// PU2150-03 PUSH DIVERT Extended
PX_4291_Extended(
	In:= In_PX_4291_Extended,
	CFG_OKState:= 0,
	CFG_OnDlyTime:= DebounceOnTime,
	CFG_OnDlyTime:= DebounceOffTime,
	In_Sim:= 
	);

// PU2150-03 PUSH DIVERT Retracted
PX_4311_Retracted(
	In:= In_PX_4311_Retracted,
	CFG_OKState:= 0,
	CFG_OnDlyTime:= DebounceOnTime,
	CFG_OnDlyTime:= DebounceOffTime,
	In_Sim:= 
	);

// PL2140 PLOW DIVERT PISTON PROX Extended
PX_10181_Extended(
	In:= In_PX_10181_Extended,
	CFG_OKState:= 0,
	CFG_OnDlyTime:= DebounceOnTime,
	CFG_OnDlyTime:= DebounceOffTime,
	In_Sim:= 
	);

// PL2140 PLOW DIVERT Extended
PX_10211_Extended(
	In:= In_PX_10211_Extended,
	CFG_OKState:= 0,
	CFG_OnDlyTime:= DebounceOnTime,
	CFG_OnDlyTime:= DebounceOffTime,
	In_Sim:= 
	);

// PL2140 PLOW DIVERT Retracted
PX_10231_Retracted(
	In:= In_PX_10231_Retracted,
	CFG_OKState:= 0,
	CFG_OnDlyTime:= DebounceOnTime,
	CFG_OnDlyTime:= DebounceOffTime,
	In_Sim:= 
	);

// PI2140 PIN STOP Extended
PX_11181_Extended(
	In:= In_PX_11181_Extended,
	CFG_OKState:= 0,
	CFG_OnDlyTime:= DebounceOnTime,
	CFG_OnDlyTime:= DebounceOffTime,
	In_Sim:= 
	);

// PI2140 PIN STOP Retracted
PX_11201_Retracted(
	In:= In_PX_11201_Retracted,
	CFG_OKState:= 0,
	CFG_OnDlyTime:= DebounceOnTime,
	CFG_OnDlyTime:= DebounceOffTime,
	In_Sim:= 
	);

// GR2140-02 "D" GRIPPER Extended
PX_11291_Extended(
	In:= In_PX_11291_Extended,
	CFG_OKState:= 0,
	CFG_OnDlyTime:= DebounceOnTime,
	CFG_OnDlyTime:= DebounceOffTime,
	In_Sim:= 
	);

// GR2140-02 "D" GRIPPER Retracted
PX_11321_Retracted(
	In:= In_PX_11321_Retracted,
	CFG_OKState:= 0,
	CFG_OnDlyTime:= DebounceOnTime,
	CFG_OnDlyTime:= DebounceOffTime,
	In_Sim:= 
	);

// GR2140-01 "D" GRIPPER Extended
PX_11141_Extended(
	In:= In_PX_11141_Extended,
	CFG_OKState:= 0,
	CFG_OnDlyTime:= DebounceOnTime,
	CFG_OnDlyTime:= DebounceOffTime,
	In_Sim:= 
	);

// GR2140-01 "D" GRIPPER Retracted
PX_11161_Retracted(
	In:= In_PX_11161_Retracted,
	CFG_OKState:= 0,
	CFG_OnDlyTime:= DebounceOnTime,
	CFG_OnDlyTime:= DebounceOffTime,
	In_Sim:= 
	);

// P2130 PROX BREAK AWAY Extended
PX_12151_Extended(
	In:= In_PX_12151_Extended,
	CFG_OKState:= 0,
	CFG_OnDlyTime:= DebounceOnTime,
	CFG_OnDlyTime:= DebounceOffTime,
	In_Sim:= 
	);
	
// P3095 PROX BREAK AWAY Extended
PX_12251_Extended(
	In:= In_PX_12251_Extended,
	CFG_OKState:= 0,
	CFG_OnDlyTime:= DebounceOnTime,
	CFG_OnDlyTime:= DebounceOffTime,
	In_Sim:= 
	);

END_PROGRAM

// ---- POUs/Solenoids.TcPOU
PROGRAM Solenoids
VAR
nEquipIndex:	DINT := 0;	// Dummy Equipment Index for Non reporting equipment
//----------------------------------------2140--------------------------------------------------------------
//----------------------------------------GR2140_01--------------------------------------------------------------
   cfgGR2140_01Label:	STRING(20) :=  'GR2140_01';
   cfgGR2140_01ExtendTODetectTime:	TIME := T#5S;
   cfgGR2140_01RetractTODetectTime:	TIME := T#5S;
   GR2140_01			: FB_Solenoid_SA;
   GR2140_01_StatePB	: ST_StateCntrlPB;
	{attribute 'OPC.UA.DA' := '0'}
   GR2140_01_Status	: ST_EquipmentStatus;		// Gripper State 
//----------------------------------------GR2140_02--------------------------------------------------------------
   cfgGR2140_02Label:	STRING(20) :=  'GR2140_02';
   cfgGR2140_02ExtendTODetectTime:	TIME := T#5S;
   cfgGR2140_02RetractTODetectTime:	TIME := T#5S;
   GR2140_02			: FB_Solenoid_SA;
   GR2140_02_StatePB	: ST_StateCntrlPB;
	{attribute 'OPC.UA.DA' := '0'}
   GR2140_02_Status	: ST_EquipmentStatus;		// Gripper State 

//----------------------------------------PI2140_01--------------------------------------------------------------
   cfgPI2140_01Label:	STRING(20) :=  'PI2140_01';
   cfgPI2140_01ExtendTODetectTime:	TIME := T#5S;
   cfgPI2140_01RetractTODetectTime:	TIME := T#5S;
   PI2140_01			: FB_Solenoid_DA;
   PI2140_01_StatePB	: ST_StateCntrlPB;
	{attribute 'OPC.UA.DA' := '0'}
   PI2140_01_Status	: ST_EquipmentStatus;		// Gripper State 

//----------------------------------------PL2140_01--------------------------------------------------------------
   cfgPL2140_01Label:	STRING(20) :=  'PL2140_01';
   cfgPL2140_01ExtendTODetectTime:	TIME := T#5S;
   cfgPL2140_01RetractTODetectTime:	TIME := T#5S;
   PL2140_01			: FB_Solenoid_SA;
   PL2140_01_StatePB	: ST_StateCntrlPB;
	{attribute 'OPC.UA.DA' := '0'}
   PL2140_01_Status	: ST_EquipmentStatus;		// Gripper State 

   
//----------------------------------------2150--------------------------------------------------------------   
//----------------------------------------GR2150_01--------------------------------------------------------------
   cfgGR2150_01Label:	STRING(20) :=  'GR2150_01';
   cfgGR2150_01ExtendTODetectTime:	TIME := T#5S;
   cfgGR2150_01RetractTODetectTime:	TIME := T#5S;
   GR2150_01			: FB_Solenoid_SA;
   GR2150_01_StatePB	: ST_StateCntrlPB;
	{attribute 'OPC.UA.DA' := '0'}
   GR2150_01_Status	: ST_EquipmentStatus;		// Gripper State 

//----------------------------------------PI2150_01--------------------------------------------------------------
   cfgPI2150_01Label:	STRING(20) :=  'PI2150_01';
   cfgPI2150_01ExtendTODetectTime:	TIME := T#5S;
   cfgPI2150_01RetractTODetectTime:	TIME := T#5S;
   PI2150_01			: FB_Solenoid_SA;
   PI2150_01_StatePB	: ST_StateCntrlPB;
	{attribute 'OPC.UA.DA' := '0'}
   PI2150_01_Status	: ST_EquipmentStatus;		// Gripper State 

//----------------------------------------PU2150_01--------------------------------------------------------------
   cfgPU2150_01Label:	STRING(20) :=  'PU2150_01';
   cfgPU2150_01ExtendTODetectTime:	TIME := T#5S;
   cfgPU2150_01RetractTODetectTime:	TIME := T#5S;
   PU2150_01			: FB_Solenoid_SA;
   PU2150_01_StatePB	: ST_StateCntrlPB;
	{attribute 'OPC.UA.DA' := '0'}
   PU2150_01_Status	: ST_EquipmentStatus;		// Gripper State 

//----------------------------------------PU2150_02--------------------------------------------------------------
   cfgPU2150_02Label:	STRING(20) :=  'PU2150_02';
   cfgPU2150_02ExtendTODetectTime:	TIME := T#5S;
   cfgPU2150_02RetractTODetectTime:	TIME := T#5S;
   PU2150_02			: FB_Solenoid_SA;
   PU2150_02_StatePB	: ST_StateCntrlPB;
	{attribute 'OPC.UA.DA' := '0'}
   PU2150_02_Status	: ST_EquipmentStatus;		// Gripper State 

//----------------------------------------PU2150_03--------------------------------------------------------------
   cfgPU2150_03Label:	STRING(20) :=  'PU2150_03';
   cfgPU2150_03ExtendTODetectTime:	TIME := T#5S;
   cfgPU2150_03RetractTODetectTime:	TIME := T#5S;
   PU2150_03			: FB_Solenoid_SA;
   PU2150_03_StatePB	: ST_StateCntrlPB;
	{attribute 'OPC.UA.DA' := '0'}
   PU2150_03_Status	: ST_EquipmentStatus;		// Gripper State 

//----------------------------------------PU2150_04--------------------------------------------------------------
   cfgPU2150_04Label:	STRING(20) :=  'PU2150_04';
   cfgPU2150_04ExtendTODetectTime:	TIME := T#5S;
   cfgPU2150_04RetractTODetectTime:	TIME := T#5S;
   PU2150_04			: FB_Solenoid_SA;
   PU2150_04_StatePB	: ST_StateCntrlPB;
	{attribute 'OPC.UA.DA' := '0'}
   PU2150_04_Status	: ST_EquipmentStatus;		// Gripper State 
END_VAR

VAR PERSISTENT
//----------------------------------------GR2140_01--------------------------------------------------------------
cfgGR2140_01IntlksArry: ARRAY [0..15] OF ST_CfgEvents := [
   (Description := 'Low Air' , DeviceLabel := 'P2140' , OKState := TRUE, StopCode := E_StopCodes.LowAir),
   (Description := 'System Interlocks OK' , DeviceLabel := 'SYSTEM', OKState := TRUE, StopCode := E_StopCodes.SystemStop),
   14(())];
cfgGR2140_01EvntsArry: ARRAY [0..15] OF ST_CfgEvents := [
   (Description := 'Extend To', DeviceLabel := 'GR2140_01', LatchRequired := TRUE, OKState := FALSE, FaultWarn:= TRUE, StopCode := E_StopCodes.ActuatorTO),
   (Description := 'Retract TO', DeviceLabel := 'GR2140_01', LatchRequired := TRUE, FaultWarn:= TRUE, OKState := FALSE, StopCode := E_StopCodes.ActuatorTO),
   (Description := 'System Fault', DeviceLabel := '', OKState := TRUE, FaultWarn:= TRUE, StopCode := E_StopCodes.SystemStop),
   (Description := 'Low Air', DeviceLabel := 'P2140', OKState := TRUE, FaultWarn:= TRUE, StopCode := E_StopCodes.LowAir, EventDelay := T#100MS),
   (Description := 'System Estop', DeviceLabel := 'System', OKState := TRUE, FaultWarn:= TRUE, StopCode := E_StopCodes.SystemStop),
   (Description := 'RIO11171 Comm Fault', DeviceLabel := 'RIO11171', OKState := TRUE, FaultWarn:= TRUE, StopCode := E_StopCodes.FieldIOFLT),
   10(())];
//----------------------------------------GR2140_02--------------------------------------------------------------
cfgGR2140_02IntlksArry: ARRAY [0..15] OF ST_CfgEvents := [
   (Description := 'Low Air' , DeviceLabel := 'P2140' , OKState := TRUE, StopCode := E_StopCodes.LowAir),
   (Description := 'System Interlocks OK' , DeviceLabel := 'SYSTEM', OKState := TRUE, StopCode := E_StopCodes.SystemStop),
   14(())];
cfgGR2140_02EvntsArry: ARRAY [0..15] OF ST_CfgEvents := [
   (Description := 'Extend To', DeviceLabel := 'GR2140_02', LatchRequired := TRUE, OKState := FALSE, FaultWarn:= TRUE, StopCode := E_StopCodes.ActuatorTO),
   (Description := 'Retract TO', DeviceLabel := 'GR2140_02', LatchRequired := TRUE, FaultWarn:= TRUE, OKState := FALSE, StopCode := E_StopCodes.ActuatorTO),
   (Description := 'System Fault', DeviceLabel := '', OKState := TRUE, FaultWarn:= TRUE, StopCode := E_StopCodes.SystemStop),
   (Description := 'Low Air', DeviceLabel := 'P2140', OKState := TRUE, FaultWarn:= TRUE, StopCode := E_StopCodes.LowAir, EventDelay := T#100MS),
   (Description := 'System Estop', DeviceLabel := 'System', OKState := TRUE, FaultWarn:= TRUE, StopCode := E_StopCodes.SystemStop),
   (Description := 'RIO3171 Comm Fault', DeviceLabel := 'RIO3171', OKState := TRUE, FaultWarn:= TRUE, StopCode := E_StopCodes.FieldIOFLT),
   9(())];
//----------------------------------------PI2140_01--------------------------------------------------------------
cfgPI2140_01IntlksArry: ARRAY [0..15] OF ST_CfgEvents := [
   (Description := 'Low Air' , DeviceLabel := 'P2140' , OKState := TRUE, StopCode := E_StopCodes.LowAir),
   (Description := 'System Interlocks OK' , DeviceLabel := 'SYSTEM', OKState := TRUE, StopCode := E_StopCodes.SystemStop),
   14(())];
cfgPI2140_01EvntsArry: ARRAY [0..15] OF ST_CfgEvents := [
   (Description := 'Extend To', DeviceLabel := 'PI2140_01', LatchRequired := TRUE, OKState := FALSE, FaultWarn:= TRUE, StopCode := E_StopCodes.ActuatorTO),
   (Description := 'Retract TO', DeviceLabel := 'PI2140_01', LatchRequired := TRUE, FaultWarn:= TRUE, OKState := FALSE, StopCode := E_StopCodes.ActuatorTO),
   (Description := 'System Fault', DeviceLabel := '', OKState := TRUE, FaultWarn:= TRUE, StopCode := E_StopCodes.SystemStop),
   (Description := 'Low Air', DeviceLabel := 'P2140', OKState := TRUE, FaultWarn:= TRUE, StopCode := E_StopCodes.LowAir, EventDelay := T#100MS),
   10(())];

//----------------------------------------PL2140_01--------------------------------------------------------------
cfgPL2140_01IntlksArry: ARRAY [0..15] OF ST_CfgEvents := [
   (Description := 'Low Air' , DeviceLabel := 'P2140' , OKState := TRUE, StopCode := E_StopCodes.LowAir),
   (Description := 'System Interlocks OK' , DeviceLabel := 'SYSTEM', OKState := TRUE, StopCode := E_StopCodes.SystemStop),
   14(())];
cfgPL2140_01EvntsArry: ARRAY [0..15] OF ST_CfgEvents := [
   (Description := 'Extend To', DeviceLabel := 'PL2140_01', LatchRequired := TRUE, OKState := FALSE, FaultWarn:= TRUE, StopCode := E_StopCodes.ActuatorTO),
   (Description := 'Retract TO', DeviceLabel := 'PL2140_01', LatchRequired := TRUE, FaultWarn:= TRUE, OKState := FALSE, StopCode := E_StopCodes.ActuatorTO),
   (Description := 'System Fault', DeviceLabel := '', OKState := TRUE, FaultWarn:= TRUE, StopCode := E_StopCodes.SystemStop),
   (Description := 'Low Air', DeviceLabel := 'P2140', OKState := TRUE, FaultWarn:= TRUE, StopCode := E_StopCodes.LowAir, EventDelay := T#100MS),
   (Description := 'RIO11171 Comm Fault', DeviceLabel := 'RIO11171', OKState := TRUE, FaultWarn:= TRUE, StopCode := E_StopCodes.FieldIOFLT),
   11(())];
//----------------------------------------GR2150_01--------------------------------------------------------------
cfgGR2150_01IntlksArry: ARRAY [0..15] OF ST_CfgEvents := [
   (Description := 'Low Air' , DeviceLabel := 'P2150' , OKState := TRUE, StopCode := E_StopCodes.LowAir),
   (Description := 'System Interlocks OK' , DeviceLabel := 'SYSTEM', OKState := TRUE, StopCode := E_StopCodes.SystemStop),
   14(())];
cfgGR2150_01EvntsArry: ARRAY [0..15] OF ST_CfgEvents := [
   (Description := 'Extend To', DeviceLabel := '2150_01', LatchRequired := TRUE, OKState := FALSE, FaultWarn:= TRUE, StopCode := E_StopCodes.ActuatorTO),
   (Description := 'Retract TO', DeviceLabel := 'GR2150_01', LatchRequired := TRUE, FaultWarn:= TRUE, OKState := FALSE, StopCode := E_StopCodes.ActuatorTO),
   (Description := 'System Fault', DeviceLabel := '', OKState := TRUE, FaultWarn:= TRUE, StopCode := E_StopCodes.SystemStop),
   (Description := 'Low Air', DeviceLabel := 'P2150', OKState := TRUE, FaultWarn:= TRUE, StopCode := E_StopCodes.LowAir, EventDelay := T#100MS),
   11(())];
//----------------------------------------PI2150_01--------------------------------------------------------------
cfgPI2150_01IntlksArry: ARRAY [0..15] OF ST_CfgEvents := [
   (Description := 'Low Air' , DeviceLabel := 'P2150' , OKState := TRUE, StopCode := E_StopCodes.LowAir),
   (Description := 'System Interlocks OK' , DeviceLabel := 'SYSTEM', OKState := TRUE, StopCode := E_StopCodes.SystemStop),
   14(())];
cfgPI2150_01EvntsArry: ARRAY [0..15] OF ST_CfgEvents := [
   (Description := 'Extend To', DeviceLabel := 'PI2150_01', LatchRequired := TRUE, OKState := FALSE, FaultWarn:= TRUE, StopCode := E_StopCodes.ActuatorTO),
   (Description := 'Retract TO', DeviceLabel := 'PI2150_01', LatchRequired := TRUE, FaultWarn:= TRUE, OKState := FALSE, StopCode := E_StopCodes.ActuatorTO),
   (Description := 'System Fault', DeviceLabel := '', OKState := TRUE, FaultWarn:= TRUE, StopCode := E_StopCodes.SystemStop),
   (Description := 'Low Air', DeviceLabel := 'P2150', OKState := TRUE, FaultWarn:= TRUE, StopCode := E_StopCodes.LowAir, EventDelay := T#100MS),
   11(())];
//----------------------------------------PU2150_01--------------------------------------------------------------
cfgPU2150_01IntlksArry: ARRAY [0..15] OF ST_CfgEvents := [
   (Description := 'Low Air' , DeviceLabel := 'P2150' , OKState := TRUE, StopCode := E_StopCodes.LowAir),
   (Description := 'System Interlocks OK' , DeviceLabel := 'SYSTEM', OKState := TRUE, StopCode := E_StopCodes.SystemStop),
   14(())];
cfgPU2150_01EvntsArry: ARRAY [0..15] OF ST_CfgEvents := [
   (Description := 'Extend To', DeviceLabel := 'PU2150_01', LatchRequired := TRUE, OKState := FALSE, FaultWarn:= TRUE, StopCode := E_StopCodes.ActuatorTO),
   (Description := 'Retract TO', DeviceLabel := 'PU2150_01', LatchRequired := TRUE, FaultWarn:= TRUE, OKState := FALSE, StopCode := E_StopCodes.ActuatorTO),
   (Description := 'System Fault', DeviceLabel := '', OKState := TRUE, FaultWarn:= TRUE, StopCode := E_StopCodes.SystemStop),
   (Description := 'Low Air', DeviceLabel := 'P2150', OKState := TRUE, FaultWarn:= TRUE, StopCode := E_StopCodes.LowAir, EventDelay := T#100MS),
   (Description := 'RIO3171 Comm Fault', DeviceLabel := 'RIO3171', OKState := TRUE, FaultWarn:= TRUE, StopCode := E_StopCodes.FieldIOFLT),
   10(())];
//----------------------------------------PU2150_02--------------------------------------------------------------
cfgPU2150_02IntlksArry: ARRAY [0..15] OF ST_CfgEvents := [
   (Description := 'Low Air' , DeviceLabel := 'P2150' , OKState := TRUE, StopCode := E_StopCodes.LowAir),
   (Description := 'System Interlocks OK' , DeviceLabel := 'SYSTEM', OKState := TRUE, StopCode := E_StopCodes.SystemStop),
   14(())];
cfgPU2150_02EvntsArry: ARRAY [0..15] OF ST_CfgEvents := [
   (Description := 'Extend To', DeviceLabel := 'PU2150_02', LatchRequired := TRUE, OKState := FALSE, FaultWarn:= TRUE, StopCode := E_StopCodes.ActuatorTO),
   (Description := 'Retract TO', DeviceLabel := 'PU2150_02', LatchRequired := TRUE, FaultWarn:= TRUE, OKState := FALSE, StopCode := E_StopCodes.ActuatorTO),
   (Description := 'System Fault', DeviceLabel := '', OKState := TRUE, FaultWarn:= TRUE, StopCode := E_StopCodes.SystemStop),
   (Description := 'Low Air', DeviceLabel := 'P2150', OKState := TRUE, FaultWarn:= TRUE, StopCode := E_StopCodes.LowAir, EventDelay := T#100MS),
   (Description := 'RIO3171 Comm Fault', DeviceLabel := 'RIO3171', OKState := TRUE, FaultWarn:= TRUE, StopCode := E_StopCodes.FieldIOFLT),
   10(())];
//----------------------------------------PU2150_03--------------------------------------------------------------
cfgPU2150_03IntlksArry: ARRAY [0..15] OF ST_CfgEvents := [
   (Description := 'Low Air' , DeviceLabel := 'P2150' , OKState := TRUE, StopCode := E_StopCodes.LowAir),
   (Description := 'System Interlocks OK' , DeviceLabel := 'SYSTEM', OKState := TRUE, StopCode := E_StopCodes.SystemStop),
   14(())];
cfgPU2150_03EvntsArry: ARRAY [0..15] OF ST_CfgEvents := [
   (Description := 'Extend To', DeviceLabel := 'PU2150_03', LatchRequired := TRUE, OKState := FALSE, FaultWarn:= TRUE, StopCode := E_StopCodes.ActuatorTO),
   (Description := 'Retract TO', DeviceLabel := 'PU2150_03', LatchRequired := TRUE, FaultWarn:= TRUE, OKState := FALSE, StopCode := E_StopCodes.ActuatorTO),
   (Description := 'System Fault', DeviceLabel := '', OKState := TRUE, FaultWarn:= TRUE, StopCode := E_StopCodes.SystemStop),
   (Description := 'Low Air', DeviceLabel := 'P2150', OKState := TRUE, FaultWarn:= TRUE, StopCode := E_StopCodes.LowAir, EventDelay := T#100MS),
   (Description := 'RIO4141 Comm Fault', DeviceLabel := 'RIO4141', OKState := TRUE, FaultWarn:= TRUE, StopCode := E_StopCodes.FieldIOFLT),
   10(())];
//----------------------------------------PU2150_04--------------------------------------------------------------
cfgPU2150_04IntlksArry: ARRAY [0..15] OF ST_CfgEvents := [
   (Description := 'Low Air' , DeviceLabel := 'P2150' , OKState := TRUE, StopCode := E_StopCodes.LowAir),
   (Description := 'System Interlocks OK' , DeviceLabel := 'SYSTEM', OKState := TRUE, StopCode := E_StopCodes.SystemStop),
   14(())];
cfgPU2150_04EvntsArry: ARRAY [0..15] OF ST_CfgEvents := [
   (Description := 'Extend To', DeviceLabel := 'PU2150_04', LatchRequired := TRUE, OKState := FALSE, FaultWarn:= TRUE, StopCode := E_StopCodes.ActuatorTO),
   (Description := 'Retract TO', DeviceLabel := 'PU2150_04', LatchRequired := TRUE, FaultWarn:= TRUE, OKState := FALSE, StopCode := E_StopCodes.ActuatorTO),
   (Description := 'System Fault', DeviceLabel := '', OKState := TRUE, FaultWarn:= TRUE, StopCode := E_StopCodes.SystemStop),
   (Description := 'Low Air', DeviceLabel := 'P2150', OKState := TRUE, FaultWarn:= TRUE, StopCode := E_StopCodes.LowAir, EventDelay := T#100MS),
   (Description := 'RIO4141 Comm Fault', DeviceLabel := 'RIO4141', OKState := TRUE, FaultWarn:= TRUE, StopCode := E_StopCodes.FieldIOFLT),
   10(())];	
END_VAR

// REMOVE THIS!!!!!!
GVL_IO.SystemAirPressure := TRUE;
//----------------------------------------2140--------------------------------------------------------------
//----------------------------------------GR2140_01--------------------------------------------------------------
GR2140_01_StatePB.AutoPB := System.Cnvyr_Auto;
GR2140_01_StatePB.ManPB := System.Cnvyr_Manual;
GR2140_01_StatePB.ResetPB := System.Cnvyr_Reset;
GR2140_01_StatePB.OfflinePB := System.Cnvyr_Offline;
GR2140_01_StatePB.StopPB := System.Cnvyr_Manual;

// Initialize the Equipment Type
GR2140_01_Status.Sts_EquipmentState.EquipType := E_EquipType.Gripper_SA;

// Interlocks
GR2140_01.In_EquipIntlks.0:= GVL_IO.SystemAirPressure;
//Events
GR2140_01.In_EquipEvents.2:= SystemSafety.Safety_SystemEstopsOK;
GR2140_01.In_EquipEvents.3:= GVL_IO.SystemAirPressure;
GR2140_01.In_EquipEvents.4:= SystemSafety.Safety_SystemEstopsOK;
GR2140_01.In_EquipEvents.5:= NOT CommStatus.RIO11171_CommFault.Out;

// Function Call
GR2140_01(
   In_p_EquipStatePB:= GR2140_01_StatePB,
   In_SimActive:= System.Sys_SimActive,
   In_EquipInit:= GVL_IO.INIT,
   Cfg_UseExtedFdbc:=FALSE,
   In_P_SVReqExtend:= Singulation_Control.SortSingulation_P2140.Out_Grabber_1_Ext,
   In_EquipRtrcdFdbck := ProxSensors.PX_11161_Retracted.Out,
   In_EquipExtdFdbck := ProxSensors.PX_11141_Extended.Out,
   Cfg_EquipIndex := nEquipIndex,
   Cfg_EquipLabel := cfgGR2140_01Label,
   Cfg_EquipDefState:= System.ConvDefaultState,
   Cfg_EquipIntlksArry:= cfgGR2140_01IntlksArry,
   Cfg_EquipEvntsArry:= cfgGR2140_01EvntsArry,
   Cfg_ExtendDetectTime:= cfgGR2140_01ExtendTODetectTime,
   Cfg_RetractDetectTime:= cfgGR2140_01RetractTODetectTime,
   Sts_EquipState := GR2140_01_Status,
   Out_ExtendCrntSV => GVL_IO.GR2140_01_Extend);
//----------------------------------------GR2140_02--------------------------------------------------------------
GR2140_02_StatePB.AutoPB := System.Cnvyr_Auto;
GR2140_02_StatePB.ManPB := System.Cnvyr_Manual;
GR2140_02_StatePB.ResetPB := System.Cnvyr_Reset;
GR2140_02_StatePB.OfflinePB := System.Cnvyr_Offline;
GR2140_02_StatePB.StopPB := System.Cnvyr_Manual;

// Initialize the Equipment Type
GR2140_02_Status.Sts_EquipmentState.EquipType := E_EquipType.Gripper_SA;

// Interlocks
GR2140_02.In_EquipIntlks.0:= GVL_IO.SystemAirPressure;
//Events
GR2140_02.In_EquipEvents.2:= SystemSafety.Safety_SystemEstopsOK;
GR2140_02.In_EquipEvents.3:= GVL_IO.SystemAirPressure;
GR2140_02.In_EquipEvents.4:= SystemSafety.Safety_SystemEstopsOK;
GR2140_02.In_EquipEvents.5:= NOT CommStatus.RIO11171_CommFault.Out;

// Function Call
GR2140_02(
   In_p_EquipStatePB:= GR2140_02_StatePB,
   In_SimActive:= System.Sys_SimActive,
   In_EquipInit:= GVL_IO.INIT,
   Cfg_UseExtedFdbc:=FALSE,
   In_P_SVReqExtend:= Singulation_Control.SortSingulation_P2140.Out_Grabber_2_Ext,
   In_EquipRtrcdFdbck := ProxSensors.PX_11321_Retracted.Out,
   In_EquipExtdFdbck := ProxSensors.PX_11291_Extended.Out,
   Cfg_EquipIndex := nEquipIndex,
   Cfg_EquipLabel := cfgGR2140_02Label,
   Cfg_EquipDefState:= System.ConvDefaultState,
   Cfg_EquipIntlksArry:= cfgGR2140_02IntlksArry,
   Cfg_EquipEvntsArry:= cfgGR2140_02EvntsArry,
   Cfg_ExtendDetectTime:= cfgGR2140_02ExtendTODetectTime,
   Cfg_RetractDetectTime:= cfgGR2140_02RetractTODetectTime,
   Sts_EquipState := GR2140_02_Status,
   Out_ExtendCrntSV => GVL_IO.GR2140_02_Extend); 
//----------------------------------------PI2140_01--------------------------------------------------------------
PI2140_01_StatePB.AutoPB := System.Cnvyr_Auto;
PI2140_01_StatePB.ManPB := System.Cnvyr_Manual;
PI2140_01_StatePB.ResetPB := System.Cnvyr_Reset;
PI2140_01_StatePB.OfflinePB := System.Cnvyr_Offline;
PI2140_01_StatePB.StopPB := System.Cnvyr_Manual;

// Initialize the Equipment Type
PI2140_01_Status.Sts_EquipmentState.EquipType := E_EquipType.Gripper_DA;

// Interlocks
//PI2140_01.In_EquipIntlks.0:= GVL_IO.SystemAirPressure;
// Interlocks for downstream full when the pin stop is extended
PI2140_01.In_EquipIntlks.2:= Photoeyes.PE_8141.Out_OnOffFltrd AND ProxSensors.PX_11181_Extended.Out;
PI2140_01.In_EquipIntlks.3:= Photoeyes.PE_4161.Out_OnOffFltrd AND ProxSensors.PX_11181_Extended.Out;
//Events
PI2140_01.In_EquipEvents.2:= SystemSafety.Safety_SystemEstopsOK;
PI2140_01.In_EquipEvents.3:= GVL_IO.SystemAirPressure;
PI2140_01.In_EquipEvents.4:= SystemSafety.Safety_SystemEstopsOK;
PI2140_01.In_EquipEvents.5:= NOT CommStatus.RIO11171_CommFault.Out;

// Function Call
PI2140_01(
   In_p_EquipStatePB:= PI2140_01_StatePB,
   In_SimActive:= System.Sys_SimActive,
   In_EquipInit:= GVL_IO.INIT,
   In_P_SVReqExtend:= Singulation_Control.SortSingulation_P2140.Out_PinStop_Ext,
   In_P_SVReqRetract:= Singulation_Control.SortSingulation_P2140.Out_PinStop_Ret,
   In_EquipRtrcdFdbck := ProxSensors.PX_11201_Retracted.Out,
   In_EquipExtdFdbck := ProxSensors.PX_11181_Extended.Out,
   Cfg_EquipIndex := nEquipIndex,
   Cfg_EquipLabel := cfgPI2140_01Label,
   Cfg_EquipDefState:= System.ConvDefaultState,   Cfg_EquipIntlksArry:= cfgPI2140_01IntlksArry,
   Cfg_EquipEvntsArry:= cfgPI2140_01EvntsArry,
   Cfg_ExtendDetectTime:= cfgPI2140_01ExtendTODetectTime,
   Cfg_RetractDetectTime:= cfgPI2140_01RetractTODetectTime,
   Sts_EquipState := PI2140_01_Status,
   Out_ExtendCrntSV => GVL_IO.PI2140_01_Extend,  
   Out_RetractCrntSV => GVL_IO.PI2140_01_Retract); 
 
//----------------------------------------PL2140_01--------------------------------------------------------------
PL2140_01_StatePB.AutoPB := System.Cnvyr_Auto;
PL2140_01_StatePB.ManPB := System.Cnvyr_Manual;
PL2140_01_StatePB.ResetPB := System.Cnvyr_Reset;
PL2140_01_StatePB.OfflinePB := System.Cnvyr_Offline;
PL2140_01_StatePB.StopPB := System.Cnvyr_Manual;

// Initialize the Equipment Type
PL2140_01_Status.Sts_EquipmentState.EquipType := E_EquipType.Gripper_SA;

// Interlocks
//PL2140_01.In_EquipIntlks.0:= GVL_IO.SystemAirPressure;
PL2140_01.In_EquipIntlks.2:= Photoeyes.PE_8141.Out_OnOffFltrd;
PL2140_01.In_EquipIntlks.3:= Photoeyes.PE_4161.Out_OnOffFltrd;
//Events
PL2140_01.In_EquipEvents.2:= SystemSafety.Safety_SystemEstopsOK;
PL2140_01.In_EquipEvents.3:= GVL_IO.SystemAirPressure;
PL2140_01.In_EquipEvents.4:= SystemSafety.Safety_SystemEstopsOK;
PL2140_01.In_EquipEvents.5:= NOT CommStatus.RIO10161_CommFault.Out;
PL2140_01.In_EquipIntlks.6:= Photoeyes.PE_10151.JamDetected;

// Function Call
PL2140_01(
   In_p_EquipStatePB:= PL2140_01_StatePB,
   In_SimActive:= System.Sys_SimActive,
   In_EquipInit:= GVL_IO.INIT,
   In_P_SVReqExtend:= Sorter.aSorterDiverts_P2140[1].Output1,
   In_EquipRtrcdFdbck := ProxSensors.PX_10231_Retracted.Out,
   In_EquipExtdFdbck := ProxSensors.PX_10211_Extended.Out,
   Cfg_EquipIndex := nEquipIndex,
   Cfg_EquipLabel := cfgPL2140_01Label,
   Cfg_EquipDefState:= System.ConvDefaultState,
   Cfg_EquipIntlksArry:= cfgPL2140_01IntlksArry,
   Cfg_EquipEvntsArry:= cfgPL2140_01EvntsArry,
   Cfg_ExtendDetectTime:= cfgPL2140_01ExtendTODetectTime,
   Cfg_RetractDetectTime:= cfgPL2140_01RetractTODetectTime,
   Sts_EquipState := PL2140_01_Status,
   Out_ExtendCrntSV => GVL_IO.PL2140_01_Extend); 
//----------------------------------------GR2150_01--------------------------------------------------------------
GR2150_01_StatePB.AutoPB := System.Cnvyr_Auto;
GR2150_01_StatePB.ManPB := System.Cnvyr_Manual;
GR2150_01_StatePB.ResetPB := System.Cnvyr_Reset;
GR2150_01_StatePB.OfflinePB := System.Cnvyr_Offline;
GR2150_01_StatePB.StopPB := System.Cnvyr_Manual;

// Initialize the Equipment Type
GR2150_01_Status.Sts_EquipmentState.EquipType := E_EquipType.Gripper_SA;

// Interlocks
GR2150_01.In_EquipIntlks.0:= GVL_IO.SystemAirPressure;
//Events
GR2150_01.In_EquipEvents.2:= SystemSafety.Safety_SystemEstopsOK;
GR2150_01.In_EquipEvents.3:= GVL_IO.SystemAirPressure;
GR2150_01.In_EquipEvents.4:= SystemSafety.Safety_SystemEstopsOK;
PI2150_01.In_EquipEvents.5:= NOT CommStatus.RIO3171_CommFault.Out;

// Function Call
GR2150_01(
   In_p_EquipStatePB:= GR2150_01_StatePB,
   In_SimActive:= System.Sys_SimActive,
   In_EquipInit:= GVL_IO.INIT,
   Cfg_UseExtedFdbc:=FALSE,
   In_P_SVReqExtend:= Singulation_Control.SortSingulation_P2150.Out_Grabber_1_Ext,
   In_EquipRtrcdFdbck := ProxSensors.PX_2201_Retracted.Out,
   In_EquipExtdFdbck := ProxSensors.PX_2181_Extended.Out,
   Cfg_EquipIndex := nEquipIndex,
   Cfg_EquipLabel := cfgGR2150_01Label,
   Cfg_EquipDefState:= System.ConvDefaultState,
   Cfg_EquipIntlksArry:= cfgGR2150_01IntlksArry,
   Cfg_EquipEvntsArry:= cfgGR2150_01EvntsArry,
   Cfg_ExtendDetectTime:= cfgGR2150_01ExtendTODetectTime,
   Cfg_RetractDetectTime:= cfgGR2150_01RetractTODetectTime,
   Sts_EquipState := GR2150_01_Status,
   Out_ExtendCrntSV => GVL_IO.GR2150_01_Extend); 
//----------------------------------------PI2150_01--------------------------------------------------------------
PI2150_01_StatePB.AutoPB := System.Cnvyr_Auto;
PI2150_01_StatePB.ManPB := System.Cnvyr_Manual;
PI2150_01_StatePB.ResetPB := System.Cnvyr_Reset;
PI2150_01_StatePB.OfflinePB := System.Cnvyr_Offline;
PI2150_01_StatePB.StopPB := System.Cnvyr_Manual;

// Initialize the Equipment Type
PI2150_01_Status.Sts_EquipmentState.EquipType := E_EquipType.Gripper_SA;

// Interlocks
PI2150_01.In_EquipIntlks.0:= GVL_IO.SystemAirPressure;
//Events
PI2150_01.In_EquipEvents.2:= SystemSafety.Safety_SystemEstopsOK;
PI2150_01.In_EquipEvents.3:= GVL_IO.SystemAirPressure;
PI2150_01.In_EquipEvents.4:= SystemSafety.Safety_SystemEstopsOK;
PI2150_01.In_EquipEvents.5:= NOT CommStatus.RIO3171_CommFault.Out;

// Function Call
PI2150_01(
   In_p_EquipStatePB:= PI2150_01_StatePB,
   In_SimActive:= System.Sys_SimActive,
   In_EquipInit:= GVL_IO.INIT,
   In_P_SVReqExtend:= Singulation_Control.SortSingulation_P2150.Out_PinStop_Ext,
   In_EquipRtrcdFdbck := ProxSensors.PX_2151_Retracted.Out,
   In_EquipExtdFdbck := ProxSensors.PX_2131_Extended.Out,
   Cfg_EquipIndex := nEquipIndex,
   Cfg_EquipLabel := cfgPI2150_01Label,
   Cfg_EquipDefState:= System.ConvDefaultState,
   Cfg_EquipIntlksArry:= cfgPI2150_01IntlksArry,
   Cfg_EquipEvntsArry:= cfgPI2150_01EvntsArry,
   Cfg_ExtendDetectTime:= cfgPI2150_01ExtendTODetectTime,
   Cfg_RetractDetectTime:= cfgPI2150_01RetractTODetectTime,
   Sts_EquipState := PI2150_01_Status,
   Out_ExtendCrntSV => GVL_IO.PI2150_01_Extend); 
//----------------------------------------PU2150_01--------------------------------------------------------------
PU2150_01_StatePB.AutoPB := System.Cnvyr_Auto;
PU2150_01_StatePB.ManPB := System.Cnvyr_Manual;
PU2150_01_StatePB.ResetPB := System.Cnvyr_Reset;
PU2150_01_StatePB.OfflinePB := System.Cnvyr_Offline;
PU2150_01_StatePB.StopPB := System.Cnvyr_Manual;

// Initialize the Equipment Type
PU2150_01_Status.Sts_EquipmentState.EquipType := E_EquipType.Gripper_SA;

// Interlocks
PU2150_01.In_EquipIntlks.0:= GVL_IO.SystemAirPressure;
//Events
PU2150_01.In_EquipEvents.2:= SystemSafety.Safety_SystemEstopsOK;
PU2150_01.In_EquipEvents.3:= GVL_IO.SystemAirPressure;
PU2150_01.In_EquipEvents.4:= SystemSafety.Safety_SystemEstopsOK;
PU2150_01.In_EquipEvents.5:= NOT CommStatus.RIO3171_CommFault.Out;

// Function Call
PU2150_01(
   In_p_EquipStatePB:= PU2150_01_StatePB,
   In_SimActive:= System.Sys_SimActive,
   In_EquipInit:= GVL_IO.INIT,
   In_P_SVReqExtend:= Sorter.aSorterDiverts_P2150[1].Output1,
   In_EquipRtrcdFdbck := ProxSensors.PX_3331_Retracted.Out,
   In_EquipExtdFdbck := ProxSensors.PX_3301_Extended.Out,
   Cfg_EquipIndex := nEquipIndex,
   Cfg_EquipLabel := cfgPU2150_01Label,
   Cfg_EquipDefState:= System.ConvDefaultState,
   Cfg_EquipIntlksArry:= cfgPU2150_01IntlksArry,
   Cfg_EquipEvntsArry:= cfgPU2150_01EvntsArry,
   Cfg_ExtendDetectTime:= cfgPU2150_01ExtendTODetectTime,
   Cfg_RetractDetectTime:= cfgPU2150_01RetractTODetectTime,
   Sts_EquipState := PU2150_01_Status,
   Out_ExtendCrntSV => GVL_IO.PU2150_01_Extend); 
//----------------------------------------PU2150_02--------------------------------------------------------------
PU2150_02_StatePB.AutoPB := System.Cnvyr_Auto;
PU2150_02_StatePB.ManPB := System.Cnvyr_Manual;
PU2150_02_StatePB.ResetPB := System.Cnvyr_Reset;
PU2150_02_StatePB.OfflinePB := System.Cnvyr_Offline;
PU2150_02_StatePB.StopPB := System.Cnvyr_Manual;

// Initialize the Equipment Type
PU2150_02_Status.Sts_EquipmentState.EquipType := E_EquipType.Gripper_SA;

// Interlocks
PU2150_02.In_EquipIntlks.0:= GVL_IO.SystemAirPressure;
//Events
PU2150_02.In_EquipEvents.2:= SystemSafety.Safety_SystemEstopsOK;
PU2150_02.In_EquipEvents.3:= GVL_IO.SystemAirPressure;
PU2150_02.In_EquipEvents.4:= SystemSafety.Safety_SystemEstopsOK;
PU2150_02.In_EquipEvents.5:= NOT CommStatus.RIO3171_CommFault.Out;

// Function Call
PU2150_02(
   In_p_EquipStatePB:= PU2150_02_StatePB,
   In_SimActive:= System.Sys_SimActive,
   In_EquipInit:= GVL_IO.INIT,
   In_P_SVReqExtend:= Sorter.aSorterDiverts_P2150[2].Output1,
   In_EquipRtrcdFdbck := ProxSensors.PX_3191_Retracted.Out,
   In_EquipExtdFdbck := ProxSensors.PX_3171_Extended.Out,
   Cfg_EquipIndex := nEquipIndex,
   Cfg_EquipLabel := cfgPU2150_02Label,
   Cfg_EquipDefState:= System.ConvDefaultState,
   Cfg_EquipIntlksArry:= cfgPU2150_02IntlksArry,
   Cfg_EquipEvntsArry:= cfgPU2150_02EvntsArry,
   Cfg_ExtendDetectTime:= cfgPU2150_02ExtendTODetectTime,
   Cfg_RetractDetectTime:= cfgPU2150_02RetractTODetectTime,
   Sts_EquipState := PU2150_02_Status,
   Out_ExtendCrntSV => GVL_IO.PU2150_02_Extend); 
//----------------------------------------PU2150_03--------------------------------------------------------------
PU2150_03_StatePB.AutoPB := System.Cnvyr_Auto;
PU2150_03_StatePB.ManPB := System.Cnvyr_Manual;
PU2150_03_StatePB.ResetPB := System.Cnvyr_Reset;
PU2150_03_StatePB.OfflinePB := System.Cnvyr_Offline;
PU2150_03_StatePB.StopPB := System.Cnvyr_Manual;

// Initialize the Equipment Type
PU2150_03_Status.Sts_EquipmentState.EquipType := E_EquipType.Gripper_SA;

// Interlocks
PU2150_03.In_EquipIntlks.0:= GVL_IO.SystemAirPressure;
//Events
PU2150_03.In_EquipEvents.2:= SystemSafety.Safety_SystemEstopsOK;
PU2150_03.In_EquipEvents.3:= GVL_IO.SystemAirPressure;
PU2150_03.In_EquipEvents.4:= SystemSafety.Safety_SystemEstopsOK;
PU2150_03.In_EquipEvents.5:= NOT CommStatus.RIO4141_CommFault.Out;

// Function Call
PU2150_03(
   In_p_EquipStatePB:= PU2150_03_StatePB,
   In_SimActive:= System.Sys_SimActive,
   In_EquipInit:= GVL_IO.INIT,
   In_P_SVReqExtend:= Sorter.aSorterDiverts_P2150[3].Output1,
   In_EquipRtrcdFdbck := ProxSensors.PX_4311_Retracted.Out,
   In_EquipExtdFdbck := ProxSensors.PX_4291_Extended.Out,
   Cfg_EquipIndex := nEquipIndex,
   Cfg_EquipLabel := cfgPU2150_03Label,
   Cfg_EquipDefState:= System.ConvDefaultState,
   Cfg_EquipIntlksArry:= cfgPU2150_03IntlksArry,
   Cfg_EquipEvntsArry:= cfgPU2150_03EvntsArry,
   Cfg_ExtendDetectTime:= cfgPU2150_03ExtendTODetectTime,
   Cfg_RetractDetectTime:= cfgPU2150_03RetractTODetectTime,
   Sts_EquipState := PU2150_03_Status,
   Out_ExtendCrntSV => GVL_IO.PU2150_03_Extend);
//----------------------------------------PU2150_04--------------------------------------------------------------
PU2150_04_StatePB.AutoPB := System.Cnvyr_Auto;
PU2150_04_StatePB.ManPB := System.Cnvyr_Manual;
PU2150_04_StatePB.ResetPB := System.Cnvyr_Reset;
PU2150_04_StatePB.OfflinePB := System.Cnvyr_Offline;
PU2150_04_StatePB.StopPB := System.Cnvyr_Manual;

// Initialize the Equipment Type
PU2150_04_Status.Sts_EquipmentState.EquipType := E_EquipType.Gripper_SA;

// Interlocks
PU2150_04.In_EquipIntlks.0:= GVL_IO.SystemAirPressure;
//Events
PU2150_04.In_EquipEvents.2:= SystemSafety.Safety_SystemEstopsOK;
PU2150_04.In_EquipEvents.3:= GVL_IO.SystemAirPressure;
PU2150_04.In_EquipEvents.4:= SystemSafety.Safety_SystemEstopsOK;
PU2150_04.In_EquipEvents.5:= NOT CommStatus.RIO4141_CommFault.Out;

// Function Call
PU2150_04(
   In_p_EquipStatePB:= PU2150_04_StatePB,
   In_SimActive:= System.Sys_SimActive,
   In_EquipInit:= GVL_IO.INIT,
   In_P_SVReqExtend:= Sorter.aSorterDiverts_P2150[4].Output1,
   In_EquipRtrcdFdbck := ProxSensors.PX_4171_Retracted.Out,
   In_EquipExtdFdbck := ProxSensors.PX_4151_Extended.Out,
   Cfg_EquipIndex := nEquipIndex,
   Cfg_EquipLabel := cfgPU2150_04Label,
   Cfg_EquipDefState:= System.ConvDefaultState,
   Cfg_EquipIntlksArry:= cfgPU2150_04IntlksArry,
   Cfg_EquipEvntsArry:= cfgPU2150_04EvntsArry,
   Cfg_ExtendDetectTime:= cfgPU2150_04ExtendTODetectTime,
   Cfg_RetractDetectTime:= cfgPU2150_04RetractTODetectTime,
   Sts_EquipState := PU2150_04_Status,
   Out_ExtendCrntSV => GVL_IO.PU2150_04_Extend);

END_PROGRAM

// ---- FunctionBlocks/Solenoids/Functions/FB_Solenoid_SA.TcPOU
FUNCTION_BLOCK FB_Solenoid_SA

(* Single-Acting solenoid Set up,
	Uses Interlocks. No common interlocks
	Doesn't use Start Conditions or the horn delay  
	Uses Events and has 5 that can be uassigned that are location specific and a common events for the Actuator Extended/Retracted Time-out faults 

	Regardless of the travel of the actuator, the following define the extended and retracted positions
		Extended is the position expected when the solenoid valve is actuated
		Retracted is the position expected when the solenoid valve is resting
*)

VAR_IN_OUT
	CFG_EquipIndex				: DINT;	// Index used for local Equipment status array
	{attribute 'OPC.UA.DA' := '1'}
	Sts_EquipState					: ST_EquipmentStatus;		// State Status
//	In_EquipEvents					: UINT;		// Event that is specific to the instance of the solenoid/actuator
//	In_EquipIntlks					: UINT;		// Interlock that is specific to the instance of the solenoid/actuator
END_VAR
VAR_INPUT
	{attribute 'OPC.UA.DA' := '1'}
	In_o_EquipStatePB				: ST_StateCntrlPB;		// Hmi push buttons to change states
	In_p_EquipStatePB				: ST_StateCntrlPB;		// programming to change states
	In_P_SVReqExtend			: BOOL;		// Input to extend actuator if in auto and conditions are met
	In_SimActive				: BOOL;
	In_EquipInit					: BOOL;		// Initialise;
	{attribute 'OPC.UA.DA' := '1'}
	In_EquipExtdFdbck			: BOOL := FALSE;	// Actuator Extended Feedback (1 = Extended)
	{attribute 'OPC.UA.DA' := '1'}
	In_EquipRtrcdFdbck			: BOOL := FALSE;	// Actuator Retracted Feedback (1 = Retracted)
	Cfg_EquipDefState				: E_StateCntrl;
	{attribute 'OPC.UA.DA' := '1'}
	Cfg_EquipLabel					: STRING(20);		// Label of the Solenoid
	Cfg_UseExtedFdbc			: BOOL := FALSE;	// Use Feedback from actuator for Extended state, otherwise, use output 

	// Events
	In_EquipEvents					: UINT;		// Event that is specific to the instance of the solenoid/actuator
	
	{attribute 'OPC.UA.DA' := '0'}
	Cfg_EquipEvntsArry				: ARRAY [0..15] OF ST_CfgEvents;
	Cfg_ExtendDetectTime		: TIME;
	Cfg_RetractDetectTime		: TIME;
	
	// Interlocks that can be Instance Specific
	In_EquipIntlks					: UINT;		// Interlock that is specific to the instance of the solenoid/actuator
	{attribute 'OPC.UA.DA' := '0'}
	Cfg_EquipIntlksArry			: ARRAY [0..15] OF ST_CfgEvents;		// Descriptions of the Interlock 
	
END_VAR
VAR_OUTPUT
	{attribute 'OPC.UA.DA' := '1'}
	Out_ExtendCrntSV			: BOOL;		// Extend command for the current solenoid/actuator
	{attribute 'OPC.UA.DA' := '1'}
	Sts_ExtendCrntSV			: BOOL;		// Status showing that current solenoid/actuator is extended/extending
	{attribute 'OPC.UA.DA' := '1'}
	Sts_All_Intlks_OK			: BOOL;		// Status bit to show that all interloks are good to Run 
	{attribute 'OPC.UA.DA' := '1'}
	Sts_FaultActive				: BOOL;	// Status Bit Showing that a fault is present (0= No Active Faults, 1= Fault Active)
	{attribute 'OPC.UA.DA' := '1'}
	Sts_WarnActive				: BOOL;	// Status Bit Showing that a warning is present (0= No Active Warnings, 1= Warning Active)
	{attribute 'OPC.UA.DA' := '1'}
	Sts_All_Evnts_OK			: BOOL;		// Status Bit Showing that ALL Events are OK to RUN (0= Event Present, 1= OK to Run)
	{attribute 'OPC.UA.DA' := '1'}
	Sts_IntlksArry				: ARRAY[0..15] OF ST_EventSts;		// Interlock status 0 to 15 Input
	{attribute 'OPC.UA.DA' := '1'}
	Sts_FaultsArry				: ARRAY[0..15] OF ST_EventSts;	// Status of each Fault Event State (0= OFF, 1=ON)
	{attribute 'OPC.UA.DA' := '1'}
	Sts_WarnsArry				: ARRAY[0..15] OF ST_EventSts;		// Status of each Warning Event State (0= OFF, 1=ON)
	{attribute 'OPC.UA.DA' := '0'}
	Sts_EvntsArry				: ARRAY[0..15] OF ST_EventSts; 	// Status of each Event State (0= OFF, 1=ON)
END_VAR
VAR
	{attribute 'OPC.UA.DA' := '0'}
	SV_fbIntrlks				: FB_Intlks_Latch;
	SV_IntlksArry				: ARRAY[0..15] OF BOOL;
	{attribute 'OPC.UA.DA' := '0'}
	SV_fbEquipCntrl				: FB_EquipCntrl;
	{attribute 'OPC.UA.DA' := '0'}
	SV_EventManager				: FB_EventMngr;
	SV_ExtendFault				: FB_JamDetect;			// This FB can also detect when it takes to long to extend an actuator
	SV_RetractFault				: FB_JamDetect;			// This FB can also detect when it takes to long to retract an actuator
	SV_EventArry				: ARRAY[0..15] OF BOOL;
	
	SV_LatchIgnore				: BOOL := FALSE;		// Put as a place holder for ease of future use
	SV_LatchReset				: BOOL := FALSE;		//Put as a place holder for ease of future use
	SV_IntlkBypassed			: ARRAY [0..15] OF BOOL;		//Put as a place holder for ease of future use
	SV_MoveEnabled				: BOOL;					// TRUE = Enable the SV/Actuator to operate
	SV_StartEnabled				: BOOL;					// TRUE = Start Motion for SV/actuator

END_VAR

// Set Up Common Single-Acting solenoid Interlocks and inputs for interlocks that are specific for the configuration instance
SV_IntlksArry[0] := In_EquipIntlks.0;
SV_IntlksArry[1] := System.SysIntlksAllOk; 
SV_IntlksArry[2] := In_EquipIntlks.2;
SV_IntlksArry[3] := In_EquipIntlks.3;
SV_IntlksArry[4] := In_EquipIntlks.4;
SV_IntlksArry[5] := In_EquipIntlks.5;
SV_IntlksArry[6] := In_EquipIntlks.6;
SV_IntlksArry[7] := In_EquipIntlks.7;
SV_IntlksArry[8] := In_EquipIntlks.8;
SV_IntlksArry[9] := In_EquipIntlks.9; 
SV_IntlksArry[10] := In_EquipIntlks.10;
SV_IntlksArry[11] := In_EquipIntlks.11;
SV_IntlksArry[12] := In_EquipIntlks.12;
SV_IntlksArry[13] := In_EquipIntlks.13;
SV_IntlksArry[14] := In_EquipIntlks.14;
SV_IntlksArry[15] := In_EquipIntlks.15;

In_EquipIntlks:=0;
	
// Call Interlock block
SV_fbIntrlks(
	In_Intlks:= SV_IntlksArry,
	CFG_IntlksArry:= Cfg_EquipIntlksArry, 
	HMI_LatchIgnore:= SV_LatchIgnore, 
	HMI_LatchReset:= SV_LatchReset, 
	All_Intlk_OK=> Sts_All_Intlks_OK, 
	STS_Intlks=> Sts_IntlksArry);
	
// Set Up Common Solenoid Events and inputs for events that are specific for the configuration instance
SV_EventArry[0]:= SV_ExtendFault.JamDetected;	// Even though this is a JamDetected output, it is really a Extend time-out fault
SV_EventArry[1]:= SV_RetractFault.JamDetected;	// Even though this is a JamDetected output, it is really a retract time-out fault
SV_EventArry[2]:= In_EquipEvents.2;
SV_EventArry[3]:= In_EquipEvents.3;
SV_EventArry[4]:= In_EquipEvents.4;
SV_EventArry[5]:= In_EquipEvents.5;
SV_EventArry[6]:= In_EquipEvents.6;
SV_EventArry[7]:= In_EquipEvents.7;
SV_EventArry[8]:= In_EquipEvents.8;
SV_EventArry[9]:= In_EquipEvents.9;
SV_EventArry[10]:= In_EquipEvents.10;
SV_EventArry[11]:= In_EquipEvents.11;
SV_EventArry[12]:= In_EquipEvents.12;
SV_EventArry[13]:= In_EquipEvents.13;
SV_EventArry[14]:= In_EquipEvents.14;
SV_EventArry[15]:= In_EquipEvents.15;

//In_EquipEvents:=0;

// Event Manager
SV_EventManager(
	sEquipStateCntrlSts := Sts_EquipState.Sts_EquipmentState,
	In_EventsArry := SV_EventArry ,  
	CFG_EvntsArry:= Cfg_EquipEvntsArry, 
	HMI_LatchReset:= In_o_EquipStatePB.ResetPB OR In_p_EquipStatePB.ResetPB,
	Out_FaultActive=> Sts_FaultActive, 
	Out_WarnActive=> Sts_WarnActive, 
	Sts_All_Evnts_OK=> Sts_All_Evnts_OK, 
	Sts_FaultsArry=> Sts_FaultsArry, 
	Sts_WarnsArry=> Sts_WarnsArry, 
	Sts_EvntsArry=> Sts_EvntsArry);
	
(*
	Set up individual Events that are common for this configuration
 	For the Extend Fault, use one of two conditions
		1 - If the SV is configured to use Extended feedback, check the input
		2 - If the SV is not configured to use Extedned feedback, check that the output is on and the retracted input is not on
*)
SV_ExtendFault.In_PE := ((Cfg_UseExtedFdbc AND NOT In_EquipExtdFdbck)
					OR (NOT Cfg_UseExtedFdbc AND (Out_ExtendCrntSV AND In_EquipRtrcdFdbck)))
					AND NOT Sts_EquipState.Sts_EquipmentState.StsOffline
					AND NOT In_o_EquipStatePB.ResetPB
					AND NOT In_p_EquipStatePB.ResetPB;
SV_ExtendFault(
	In_Status:= Out_ExtendCrntSV,
	CFG_PEOKState:= 0, 
	JamDetTime:= cfg_ExtendDetectTime);
	
(*
 	For the Retract Fault, use the following condition
		Output is off and the actuator is not in the retracted condition
*)
SV_RetractFault.In_PE := NOT Out_ExtendCrntSV
					AND NOT In_EquipRtrcdFdbck
					AND NOT Sts_EquipState.Sts_EquipmentState.StsOffline
					AND NOT In_o_EquipStatePB.ResetPB
					AND NOT In_p_EquipStatePB.ResetPB;
SV_RetractFault(
	In_Status:= NOT Out_ExtendCrntSV,
	CFG_PEOKState:= 0, 
	JamDetTime:= cfg_RetractDetectTime);

//Call Equipment FB to control current SV/Actuator	
SV_fbEquipCntrl(
	CFG_EquipIndex := cfg_EquipIndex,
	CFG_EquipLabel := Cfg_EquipLabel,
	CFG_UseStrtCnd:= FALSE, 
	CFG_UseIntrlks:= TRUE, 
	CFG_UseHrnDly:= FALSE, 
	CFG_EquipDefState:= Cfg_EquipDefState, 
	In_IntlksOK:= Sts_All_Intlks_OK, 
	In_SimActive:= In_SimActive, 
	In_Init:= In_EquipInit, 
	o_EquipStatePB:= In_o_EquipStatePB, 
	p_EquipStatePB:= In_p_EquipStatePB, 
	P_EquipReqRun:= In_P_SVReqExtend, 
	In_EquipFaults:= Sts_FaultActive, 
	Out_EquipRun=> , 
	Out_Horn=> , 
	Sts_EquipState:= Sts_EquipState.Sts_EquipmentState);	

// Process the SV_MoveEnabled signal
SV_MoveEnabled := SV_fbEquipCntrl.Out_EquipRun;

SV_StartEnabled := SV_MoveEnabled;	

// Actuate the SV based on the results of the Equipment Control state
IF Sts_EquipState.Sts_EquipmentState.CrntState = E_StateCntrl.stAuto THEN
	IF (In_P_SVReqExtend )
	   THEN
		Out_ExtendCrntSV := SV_StartEnabled;
		// Set Solenoid Actuation Status
		Sts_ExtendCrntSV := (Out_ExtendCrntSV) OR (In_SimActive AND SV_fbEquipCntrl.RunApproved);
	ELSE
		Out_ExtendCrntSV := FALSE;
		// Set Solenoid Actuation Status
		Sts_ExtendCrntSV := FALSE;
	END_IF
ELSE
	IF (In_o_EquipStatePB.ManExtendPB)
	   THEN
		Out_ExtendCrntSV := SV_StartEnabled;
		// Set Solenoid Actuation Status
		Sts_ExtendCrntSV := (Out_ExtendCrntSV) OR (In_SimActive AND SV_fbEquipCntrl.RunApproved);
	ELSE
		Out_ExtendCrntSV := FALSE;
		// Set Solenoid Actuation Status
		Sts_ExtendCrntSV := FALSE;
	END_IF
END_IF

// Turn OFF Extend and Retract when a stop is issued
IF In_p_EquipStatePB.StopPB OR In_o_EquipStatePB.StopPB OR Sts_FaultActive THEN
	Out_ExtendCrntSV := FALSE;
	Sts_ExtendCrntSV := FALSE;
END_IF

// Capture the Operation state of the Solenoid/actuator
IF Sts_ExtendCrntSV THEN
	// Solenoid Actuating/Entending
	Sts_EquipState.Sts_EquipmentState.CrntOperState := E_OperStateCntrl.extending;
	// Solenoid Extended
	IF (Cfg_UseExtedFdbc AND In_EquipExtdFdbck) OR (NOT Cfg_UseExtedFdbc AND (Out_ExtendCrntSV AND NOT In_EquipRtrcdFdbck)) THEN
		Sts_EquipState.Sts_EquipmentState.CrntOperState := E_OperStateCntrl.extended;
	END_IF
ELSE
	// Solenoid Retracting
	Sts_EquipState.Sts_EquipmentState.CrntOperState := E_OperStateCntrl.retracting;
	// Solenoid Retracted
	IF In_EquipRtrcdFdbck THEN
		Sts_EquipState.Sts_EquipmentState.CrntOperState := E_OperStateCntrl.retracted;
	END_IF
END_IF
IF NOT Sts_ExtendCrntSV
   AND NOT In_EquipRtrcdFdbck
   AND NOT (Cfg_UseExtedFdbc AND In_EquipExtdFdbck) OR (NOT Cfg_UseExtedFdbc AND (Out_ExtendCrntSV AND NOT In_EquipRtrcdFdbck)) 
   THEN
	Sts_EquipState.Sts_EquipmentState.CrntOperState := E_OperStateCntrl.unknown;
END_IF
// Solenoid control and state
CASE Sts_EquipState.Sts_EquipmentState.CrntOperState OF
	E_OperStateCntrl.extended:
			Sts_EquipState.Sts_IsExtended := TRUE;
			Sts_EquipState.Sts_IsExtending := FALSE;
			Sts_EquipState.Sts_IsRetracted := FALSE;
			Sts_EquipState.Sts_IsRetracting := FALSE;
	E_OperStateCntrl.extending:
			Sts_EquipState.Sts_IsExtended := FALSE;
			Sts_EquipState.Sts_IsExtending := TRUE;
			Sts_EquipState.Sts_IsRetracted := FALSE;
			Sts_EquipState.Sts_IsRetracting := FALSE;
	E_OperStateCntrl.retracted:
			Sts_EquipState.Sts_IsExtended := FALSE;
			Sts_EquipState.Sts_IsExtending := FALSE;
			Sts_EquipState.Sts_IsRetracted := TRUE;
			Sts_EquipState.Sts_IsRetracting := FALSE;
	E_OperStateCntrl.retracting:
			Sts_EquipState.Sts_IsExtended := FALSE;
			Sts_EquipState.Sts_IsExtending := FALSE;
			Sts_EquipState.Sts_IsRetracted := FALSE;
			Sts_EquipState.Sts_IsRetracting := TRUE;
END_CASE

// Populate the Sts Output Variables
Sts_EquipState.Sts_All_Intlks_OK  := Sts_All_Intlks_OK;
Sts_EquipState.Sts_All_Evnts_OK  := Sts_All_Evnts_OK;
Sts_EquipState.Sts_FaultActive := Sts_FaultActive;
Sts_EquipState.Sts_WarnActive := Sts_WarnActive;

END_FUNCTION_BLOCK

// ---- FunctionBlocks/Solenoids/Functions/FB_Solenoid_DA.TcPOU
FUNCTION_BLOCK FB_Solenoid_DA

(* Double-Acting solenoid Set up,
	Uses Interlocks. No common interlocks
	Doesn't use Start Conditions or the horn delay  
	Uses Events and has 5 that can be uassigned that are location specific and a common events for the Actuator Extended/Retracted Time-out faults 

	Regardless of the travel of the actuator, the following define the extended and retracted positions
		Extended is the position expected when the solenoid valve is actuated
		Retracted is the position expected when the solenoid valve is resting
*)

VAR_IN_OUT
	CFG_EquipIndex				: DINT;	// Index used for local Equipment status array
	{attribute 'OPC.UA.DA' := '1'}
	Sts_EquipState					: ST_EquipmentStatus;		// State Status
//	In_EquipEvents					: UINT;		// Event that is specific to the instance of the solenoid/actuator
//	In_EquipIntlks					: UINT;		// Interlock that is specific to the instance of the solenoid/actuator
END_VAR
VAR_INPUT
	{attribute 'OPC.UA.DA' := '1'}
	In_o_EquipStatePB				: ST_StateCntrlPB;		// Hmi push buttons to change states
	In_p_EquipStatePB				: ST_StateCntrlPB;		// programming to change states
	In_P_SVReqExtend			: BOOL;		// Input to extend actuator if in auto and conditions are met
	In_P_SVReqRetract			: BOOL;		// Input to retract actuator if in auto and conditions are met
	In_SimActive				: BOOL;
	In_EquipInit					: BOOL;		// Initialise;
	{attribute 'OPC.UA.DA' := '1'}
	In_EquipExtdFdbck			: BOOL := FALSE;	// Actuator Extended Feedback (1 = Extended)
	{attribute 'OPC.UA.DA' := '1'}
	In_EquipRtrcdFdbck			: BOOL := FALSE;	// Actuator Retracted Feedback (1 = Retracted)
	Cfg_EquipDefState				: E_StateCntrl;
	{attribute 'OPC.UA.DA' := '1'}
	Cfg_EquipLabel					: STRING(20);		// Label of the Solenoid
	Cfg_UseExtedFdbc			: BOOL := FALSE;	// Use Feedback from actuator for Extended state, otherwise, use output 

	// Events
	// This is the system interlock, but could be something different
	In_EquipEvents					: UINT;		// Event that is specific to the instance of the solenoid/actuator
	
	{attribute 'OPC.UA.DA' := '0'}
	Cfg_EquipEvntsArry				: ARRAY [0..15] OF ST_CfgEvents;
	Cfg_ExtendDetectTime		: TIME;
	Cfg_RetractDetectTime		: TIME;
	
	// Interlocks that can be Instance Specific
	In_EquipIntlks					: UINT;		// Interlock that is specific to the instance of the solenoid/actuator
	{attribute 'OPC.UA.DA' := '0'}
	Cfg_EquipIntlksArry			: ARRAY [0..15] OF ST_CfgEvents;		// Descriptions of the Interlock 
	
END_VAR
VAR_OUTPUT
	{attribute 'OPC.UA.DA' := '1'}
	Out_ExtendCrntSV			: BOOL;		// Extend command for the current solenoid/actuator
	{attribute 'OPC.UA.DA' := '1'}
	Sts_ExtendCrntSV			: BOOL;		// Status showing that current solenoid/actuator is extended/extending
	{attribute 'OPC.UA.DA' := '1'}
	Out_RetractCrntSV			: BOOL;		// Retract command for the current solenoid/actuator
	{attribute 'OPC.UA.DA' := '1'}
	Sts_RetractCrntSV			: BOOL;		// Status showing that current solenoid/actuator is retracteded/retractinging
	{attribute 'OPC.UA.DA' := '1'}
	Sts_All_Intlks_OK			: BOOL;		// Status bit to show that all interloks are good to Run 
	{attribute 'OPC.UA.DA' := '1'}
	Sts_FaultActive				: BOOL;	// Status Bit Showing that a fault is present (0= No Active Faults, 1= Fault Active)
	{attribute 'OPC.UA.DA' := '1'}
	Sts_WarnActive				: BOOL;	// Status Bit Showing that a warning is present (0= No Active Warnings, 1= Warning Active)
	{attribute 'OPC.UA.DA' := '1'}
	Sts_All_Evnts_OK			: BOOL;		// Status Bit Showing that ALL Events are OK to RUN (0= Event Present, 1= OK to Run)
	{attribute 'OPC.UA.DA' := '1'}
	Sts_IntlksArry				: ARRAY[0..15] OF ST_EventSts;		// Interlock status 0 to 15 Input
	{attribute 'OPC.UA.DA' := '1'}
	Sts_FaultsArry				: ARRAY[0..15] OF ST_EventSts;	// Status of each Fault Event State (0= OFF, 1=ON)
	{attribute 'OPC.UA.DA' := '1'}
	Sts_WarnsArry				: ARRAY[0..15] OF ST_EventSts;		// Status of each Warning Event State (0= OFF, 1=ON)
	{attribute 'OPC.UA.DA' := '0'}
	Sts_EvntsArry				: ARRAY[0..15] OF ST_EventSts; 	// Status of each Event State (0= OFF, 1=ON)
END_VAR
VAR
	{attribute 'OPC.UA.DA' := '0'}
	SV_fbIntrlks				: FB_Intlks_Latch;
	SV_IntlksArry				: ARRAY[0..15] OF BOOL;
	{attribute 'OPC.UA.DA' := '0'}
	SV_fbEquipCntrl				: FB_EquipCntrl;
	{attribute 'OPC.UA.DA' := '0'}
	SV_EventManager				: FB_EventMngr;
	SV_ExtendFault				: FB_JamDetect;			// This FB can also detect when it takes to long to extend an actuator
	SV_RetractFault				: FB_JamDetect;			// This FB can also detect when it takes to long to retract an actuator
	SV_EventArry				: ARRAY[0..15] OF BOOL;
	
	SV_LatchIgnore				: BOOL := FALSE;		// Put as a place holder for ease of future use
	SV_LatchReset				: BOOL := FALSE;		//Put as a place holder for ease of future use
	SV_IntlkBypassed			: ARRAY [0..15] OF BOOL;		//Put as a place holder for ease of future use
	SV_MoveEnabled				: BOOL;					// TRUE = Enable the SV/Actuator to operate
	SV_StartEnabled				: BOOL;					// TRUE = Start Motion for SV/actuator

END_VAR

// Set Up Common Single-Acting solenoid Interlocks and inputs for interlocks that are specific for the configuration instance
SV_IntlksArry[0] := In_EquipIntlks.0;
SV_IntlksArry[1] := System.SysIntlksAllOk; 
SV_IntlksArry[2] := In_EquipIntlks.2;
SV_IntlksArry[3] := In_EquipIntlks.3;
SV_IntlksArry[4] := In_EquipIntlks.4;
SV_IntlksArry[5] := In_EquipIntlks.5;
SV_IntlksArry[6] := In_EquipIntlks.6;
SV_IntlksArry[7] := In_EquipIntlks.7;
SV_IntlksArry[8] := In_EquipIntlks.8;
SV_IntlksArry[9] := In_EquipIntlks.9; 
SV_IntlksArry[10] := In_EquipIntlks.10;
SV_IntlksArry[11] := In_EquipIntlks.11;
SV_IntlksArry[12] := In_EquipIntlks.12;
SV_IntlksArry[13] := In_EquipIntlks.13;
SV_IntlksArry[14] := In_EquipIntlks.14;
SV_IntlksArry[15] := In_EquipIntlks.15;
	
In_EquipIntlks:= 0;

// Call Interlock block
SV_fbIntrlks(
	In_Intlks:= SV_IntlksArry,
	CFG_IntlksArry:= Cfg_EquipIntlksArry, 
	HMI_LatchIgnore:= SV_LatchIgnore, 
	HMI_LatchReset:= SV_LatchReset, 
	All_Intlk_OK=> Sts_All_Intlks_OK, 
	STS_Intlks=> Sts_IntlksArry);
	
// Set Up Common Solenoid Events and inputs for events that are specific for the configuration instance
SV_EventArry[0]:= SV_ExtendFault.JamDetected;	// Even though this is a JamDetected output, it is really a Extend time-out fault
SV_EventArry[1]:= SV_RetractFault.JamDetected;	// Even though this is a JamDetected output, it is really a retract time-out fault
SV_EventArry[2]:= In_EquipEvents.2;
SV_EventArry[3]:= In_EquipEvents.3;
SV_EventArry[4]:= In_EquipEvents.4;
SV_EventArry[5]:= In_EquipEvents.5;
SV_EventArry[6]:= In_EquipEvents.6;
SV_EventArry[7]:= In_EquipEvents.7;
SV_EventArry[8]:= In_EquipEvents.8;
SV_EventArry[9]:= In_EquipEvents.9;
SV_EventArry[10]:= In_EquipEvents.10;
SV_EventArry[11]:= In_EquipEvents.11;
SV_EventArry[12]:= In_EquipEvents.12;
SV_EventArry[13]:= In_EquipEvents.13;
SV_EventArry[14]:= In_EquipEvents.14;
SV_EventArry[15]:= In_EquipEvents.15;

//In_EquipEvents:=0;

// Event Manager
SV_EventManager(
	sEquipStateCntrlSts := Sts_EquipState.Sts_EquipmentState,
	In_EventsArry := SV_EventArry ,  
	CFG_EvntsArry:= Cfg_EquipEvntsArry, 
	HMI_LatchReset:= In_o_EquipStatePB.ResetPB OR In_p_EquipStatePB.ResetPB,
	Out_FaultActive=> Sts_FaultActive, 
	Out_WarnActive=> Sts_WarnActive, 
	Sts_All_Evnts_OK=> Sts_All_Evnts_OK, 
	Sts_FaultsArry=> Sts_FaultsArry, 
	Sts_WarnsArry=> Sts_WarnsArry, 
	Sts_EvntsArry=> Sts_EvntsArry);
	
(*
	Set up individual Events that are common for this configuration
 	For the Extend Fault, use one of two conditions
		1 - If the SV is configured to use Extended feedback, check the input
		2 - If the SV is not configured to use Extedned feedback, check that the output is on and the retracted input is not on
*)
SV_ExtendFault.In_PE := ((Cfg_UseExtedFdbc AND NOT In_EquipExtdFdbck)
					OR (NOT Cfg_UseExtedFdbc AND (Out_ExtendCrntSV AND In_EquipRtrcdFdbck)))
					AND NOT Sts_EquipState.Sts_EquipmentState.StsOffline
					AND NOT In_o_EquipStatePB.ResetPB
					AND NOT In_p_EquipStatePB.ResetPB;
SV_ExtendFault(
	In_Status:= Out_ExtendCrntSV,
	CFG_PEOKState:= 0, 
	JamDetTime:= cfg_ExtendDetectTime);
	
(*
 	For the Retract Fault, use the following condition
		Retracted Output is ON and the actuator is not in the retracted condition
*)
SV_RetractFault.In_PE := Out_RetractCrntSV
				AND NOT In_EquipRtrcdFdbck
				AND NOT Sts_EquipState.Sts_EquipmentState.StsOffline
				AND NOT In_o_EquipStatePB.ResetPB
				AND NOT In_p_EquipStatePB.ResetPB;
SV_RetractFault(
	In_Status:= Out_RetractCrntSV,
	CFG_PEOKState:= 0, 
	JamDetTime:= cfg_RetractDetectTime);

//Call Equipment FB to control current SV/Actuator	
// XOR the Extend and Retract. The interlocks/events must be prefixed with the extend or retract command 
SV_fbEquipCntrl(
	CFG_EquipIndex := cfg_EquipIndex,
	CFG_EquipLabel := Cfg_EquipLabel,
	CFG_UseStrtCnd:= FALSE, 
	CFG_UseIntrlks:= TRUE, 
	CFG_UseHrnDly:= FALSE, 
	CFG_EquipDefState:= Cfg_EquipDefState, 
	In_IntlksOK:= Sts_All_Intlks_OK, 
	In_SimActive:= In_SimActive, 
	In_Init:= In_EquipInit, 
	o_EquipStatePB:= In_o_EquipStatePB, 
	p_EquipStatePB:= In_p_EquipStatePB, 
	P_EquipReqRun:= In_P_SVReqExtend XOR In_P_SVReqRetract, 
	In_EquipFaults:= Sts_FaultActive, 
	Out_EquipRun=> , 
	Out_Horn=> , 
	Sts_EquipState:= Sts_EquipState.Sts_EquipmentState);	

// Process the SV_MoveEnabled signal
SV_MoveEnabled := SV_fbEquipCntrl.Out_EquipRun;

SV_StartEnabled := SV_MoveEnabled;	

// Actuate the SV based on the results of the Equipment Control state
IF Sts_EquipState.Sts_EquipmentState.CrntState = E_StateCntrl.stAuto THEN
	IF (In_P_SVReqExtend AND NOT In_P_SVReqRetract)
	   THEN
		Out_RetractCrntSV := FALSE;
		Out_ExtendCrntSV := SV_StartEnabled;
		// Set Solenoid Actuation Status
		Sts_ExtendCrntSV := (Out_ExtendCrntSV) OR (In_SimActive AND SV_fbEquipCntrl.RunApproved);
		Sts_RetractCrntSV := FALSE;
	END_IF
	IF In_P_SVReqRetract THEN
		Out_RetractCrntSV := SV_StartEnabled;
		Out_ExtendCrntSV := FALSE;
		// Set Solenoid Actuation Status
		Sts_RetractCrntSV := (Out_RetractCrntSV) OR (In_SimActive AND SV_fbEquipCntrl.RunApproved);
		Sts_ExtendCrntSV := FALSE;
	END_IF
ELSE
	IF (In_o_EquipStatePB.ManExtendPB AND NOT In_o_EquipStatePB.ManRetractPB)
	   THEN
		Out_RetractCrntSV := FALSE;
		Out_ExtendCrntSV := SV_StartEnabled;
		// Set Solenoid Actuation Status
		Sts_ExtendCrntSV := (Out_ExtendCrntSV) OR (In_SimActive AND SV_fbEquipCntrl.RunApproved);
		Sts_RetractCrntSV := FALSE;
	END_IF
	IF In_o_EquipStatePB.ManRetractPB THEN
		Out_RetractCrntSV := SV_StartEnabled;
		Out_ExtendCrntSV := FALSE;
		// Set Solenoid Actuation Status
		Sts_RetractCrntSV := (Out_RetractCrntSV) OR (In_SimActive AND SV_fbEquipCntrl.RunApproved);
		Sts_ExtendCrntSV := FALSE;
	END_IF
END_IF

// Turn OFF Extend and Retract when a stop is issued
IF In_p_EquipStatePB.StopPB OR In_o_EquipStatePB.StopPB OR Sts_FaultActive THEN
	Out_ExtendCrntSV := FALSE;
	Out_RetractCrntSV := FALSE;
	Sts_ExtendCrntSV := FALSE;
	Sts_RetractCrntSV := FALSE;
END_IF

// Capture the Operation state of the Solenoid/actuator
IF Sts_ExtendCrntSV THEN
	// Solenoid Actuating/Entending
	Sts_EquipState.Sts_EquipmentState.CrntOperState := E_OperStateCntrl.extending;
	// Solenoid Extended
	IF (Cfg_UseExtedFdbc AND In_EquipExtdFdbck) OR (NOT Cfg_UseExtedFdbc AND (Out_ExtendCrntSV AND NOT In_EquipRtrcdFdbck)) THEN
		Sts_EquipState.Sts_EquipmentState.CrntOperState := E_OperStateCntrl.extended;
	END_IF
END_IF
IF Sts_RetractCrntSV THEN
	// Solenoid Retracting
	Sts_EquipState.Sts_EquipmentState.CrntOperState := E_OperStateCntrl.retracting;
	// Solenoid Retracted
	IF In_EquipRtrcdFdbck THEN
		Sts_EquipState.Sts_EquipmentState.CrntOperState := E_OperStateCntrl.retracted;
	END_IF
END_IF
IF NOT Sts_ExtendCrntSV
   AND NOT Sts_RetractCrntSV 
   AND NOT In_EquipRtrcdFdbck
   AND NOT (Cfg_UseExtedFdbc AND In_EquipExtdFdbck) OR (NOT Cfg_UseExtedFdbc AND (Out_ExtendCrntSV AND NOT In_EquipRtrcdFdbck)) 
   THEN
	Sts_EquipState.Sts_EquipmentState.CrntOperState := E_OperStateCntrl.unknown;
END_IF
// Solenoid control and state
CASE Sts_EquipState.Sts_EquipmentState.CrntOperState OF
	E_OperStateCntrl.extended:
			Sts_EquipState.Sts_IsExtended := TRUE;
			Sts_EquipState.Sts_IsExtending := FALSE;
			Sts_EquipState.Sts_IsRetracted := FALSE;
			Sts_EquipState.Sts_IsRetracting := FALSE;
	E_OperStateCntrl.extending:
			Sts_EquipState.Sts_IsExtended := FALSE;
			Sts_EquipState.Sts_IsExtending := TRUE;
			Sts_EquipState.Sts_IsRetracted := FALSE;
			Sts_EquipState.Sts_IsRetracting := FALSE;
	E_OperStateCntrl.retracted:
			Sts_EquipState.Sts_IsExtended := FALSE;
			Sts_EquipState.Sts_IsExtending := FALSE;
			Sts_EquipState.Sts_IsRetracted := TRUE;
			Sts_EquipState.Sts_IsRetracting := FALSE;
	E_OperStateCntrl.retracting:
			Sts_EquipState.Sts_IsExtended := FALSE;
			Sts_EquipState.Sts_IsExtending := FALSE;
			Sts_EquipState.Sts_IsRetracted := FALSE;
			Sts_EquipState.Sts_IsRetracting := TRUE;
END_CASE

// Populate the Sts Output Variables
Sts_EquipState.Sts_All_Intlks_OK  := Sts_All_Intlks_OK;
Sts_EquipState.Sts_All_Evnts_OK  := Sts_All_Evnts_OK;
Sts_EquipState.Sts_FaultActive := Sts_FaultActive;
Sts_EquipState.Sts_WarnActive := Sts_WarnActive;

END_FUNCTION_BLOCK

// ---- POUs/Singulation_Control.TcPOU
PROGRAM Singulation_Control
VAR
	SortSingulation_P2140	:	FB_Singulation;
	RetryLimit_P2140		:	UINT := 1;
	ReleaseDist_P2140		:	UINT :=200;
	
	SortSingulation_P2150	:	FB_Singulation;
	RetryLimit_P2150		:	UINT := 1;
	ReleaseDist_P2150		:	UINT :=150;

END_VAR

SortSingulation_P2140.In_Hold_Request := Solenoids.PI2140_01.Sts_IntlksArry[2].Status
										OR Solenoids.PI2140_01.Sts_IntlksArry[3].Status;

SortSingulation_P2140(
	In_ConveyorRunning := Conveyors.P2140_Status.Sts_IsRunning,
	In_Grabber_1_Auto := Solenoids.GR2140_01_Status.Sts_EquipmentState.StsAuto,
	In_Grabber_1_Extended := ProxSensors.In_PX_11141_Extended,
	In_Grabber_1_Retracted := ProxSensors.In_PX_11161_Retracted,
	In_Grabber_2_Auto := Solenoids.GR2140_02_Status.Sts_EquipmentState.StsAuto,
	In_Grabber_2_Extended := ProxSensors.In_PX_11291_Extended,
	In_Grabber_2_Retracted := ProxSensors.In_PX_11321_Retracted,
	In_PinStop_Auto := Solenoids.PI2140_01_Status.Sts_EquipmentState.StsAuto,
	In_PinStop_Extended := ProxSensors.In_PX_11181_Extended,
	In_PinStop_Retracted := ProxSensors.In_PX_11201_Retracted,
	In_FaultReset := System.Cnvyr_Reset,
	In_EncoderCount := GVL_IO.ENC_9031_Raw,
	In_PE_GrabTrigger:= PhotoEyes.PE_11221.Out_OnFltrd, 
	In_PE_ToteTrigger:= PhotoEyes.PE_11191.Out_OffFltrd, 
	In_PE_ClearedTrigger:= PhotoEyes.PE_10081.Out_OffFltrd,
	Cfg_GappingDistance := ReleaseDist_P2140,
	Cfg_TimeOutTime:= T#5S,
	Cfg_RetryLimit:= RetryLimit_P2140, 
);

SortSingulation_P2150(
	In_ConveyorRunning := TRUE,
	In_Grabber_1_Auto := Solenoids.GR2150_01_Status.Sts_EquipmentState.StsAuto,
	In_Grabber_1_Extended := ProxSensors.In_PX_2181_Extended,
	In_Grabber_1_Retracted := ProxSensors.In_PX_2201_Retracted,
	In_Grabber_2_Auto := Solenoids.GR2150_01_Status.Sts_EquipmentState.StsAuto,
	In_Grabber_2_Extended := ProxSensors.In_PX_2181_Extended,
	In_Grabber_2_Retracted := ProxSensors.In_PX_2201_Retracted,
	In_PinStop_Auto := Solenoids.PI2150_01_Status.Sts_EquipmentState.StsAuto,
	In_PinStop_Extended := ProxSensors.In_PX_2131_Extended,
	In_PinStop_Retracted := ProxSensors.In_PX_2151_Retracted,
	In_FaultReset := System.Cnvyr_Reset,
	In_EncoderCount := GVL_IO.ENC_9091_Raw,
	In_PE_GrabTrigger:= PhotoEyes.PE_2331.Out_OnFltrd, 
	In_PE_ToteTrigger:= FALSE, 
	In_PE_ClearedTrigger:= PhotoEyes.PE_2301.Out_OffFltrd,
	Cfg_GappingDistance := ReleaseDist_P2150,
	Cfg_TimeOutTime:= T#5S,
	Cfg_RetryLimit:= RetryLimit_P2150, 
);

END_PROGRAM

// ---- FunctionBlocks/Singulation/FB_Singulation.TcPOU
FUNCTION_BLOCK FB_Singulation
VAR_INPUT
	{attribute 'OPC.UA.DA' := '1'}
	In_ResetState			:	BOOL;	// Clear the current functional state of the Singulator
	In_Pause				:	BOOL;
	In_FaultReset			:	BOOL;
	In_EncoderCount			:	UINT;	// Current encoder Pulse Count
	In_PE_GrabTrigger		:	BOOL;
	In_PE_ToteTrigger		:	BOOL;
	In_PE_ClearedTrigger	:	BOOL;
	In_ConveyorRunning		:	BOOL;
	
	In_Grabber_1_Auto		:	BOOL;
	In_Grabber_1_Extended	:	BOOL;
	In_Grabber_1_Retracted	:	BOOL;

	In_Grabber_2_Auto		:	BOOL;
	In_Grabber_2_Extended	:	BOOL;
	In_Grabber_2_Retracted	:	BOOL;

	In_PinStop_Auto			:	BOOL;
	In_PinStop_Extended		:	BOOL;
	In_PinStop_Retracted	:	BOOL;

	In_Hold_Request			:	BOOL;

	Cfg_GappingDistance		:	UINT;	// Distance in encoder Pulses before the next item can be released
	Cfg_TimeOutTime			:	TIME := T#3S;
	Cfg_RetryLimit			:	UINT;
END_VAR
VAR_OUTPUT
	Out_ReleaseFault		:	BOOL;

	Out_Grabber_1_Ext		:	BOOL;
	Out_Grabber_1_Ret		:	BOOL;

	Out_Grabber_2_Ext		:	BOOL;
	Out_Grabber_2_Ret		:	BOOL;

	Out_PinStop_Ext			:	BOOL;
	Out_PinStop_Ret			:	BOOL;

	Out_Homed				:	BOOL;
	Out_Ready				:	BOOL;
	Out_Running				:	BOOL;
	Out_Holding				:	BOOL;
	
	Status_Output			:	UINT;
	Status					:	UINT;
END_VAR
VAR	
	SingulatorClear			:	BOOL:= FALSE;

	RolloverDetect			:	UINT;	// Capture the last Distance when the Encoder count goes to zero
	GrabTrigger				:	R_TRIG;
	ClearedTriggerPE		:	F_TRIG;
	
	resumeFromPause   : F_TRIG;
	
	StartUp					:	BOOL := TRUE;

	ClearedPECount			:	UINT;	// Encoder Pulses when ClearedTriggerPE triggered
	ClearedDistance			:	UINT;	// Distance traveled since last item cleared
	Releasing				:	BOOL;
	ReleaseTimeOut			:	TON;
	BadReleaseCount			:	UINT;
	BadReleaseCount_Old		:	UINT;
	BadReleaseReTryTimer	:	TON;
	BadReleaseRetry			:	BOOL;

	rResetState				:	R_TRIG;

	tonHomeWait				:	TON := (PT := T#1S);
	tonReadyWait			:	TON := (PT := T#1S);
	tonRunningWait			:	TON := (PT := T#5S);

	// Extend and Retract controls
	Grabber_1_Extend		:	BOOL;
	Grabber_1_Retract		:	BOOL;

	Grabber_2_Extend		:	BOOL;
	Grabber_2_Retract		:	BOOL;

	PinStop_Extend			:	BOOL;
	PinStop_Retract			:	BOOL;
END_VAR

VAR CONSTANT
	// Output Status
	GRABBER_1_OCCUPIED		:	UINT  := 1;
	GRABBER_2_OCCUPIED		:	UINT  := 2;
	PINSTOP_OUT				:	UINT  := 3;
	
	// Singulation Status
	PAUSED					:	UINT  := 0;
	PRODUCT_PRESENT			:	UINT  := 1;
	PRODUCT_ENTERING_OCR	:	UINT  := 2;
	PRODUCT_READY_TO_PROCESS:	UINT  := 3;
	OCR_FINISHED			:	UINT  := 4;	
	PRODUCT_EXITING_OCR		:	UINT  := 5;
	RETURN_CONVEYOR_CLEARING:	UINT  := 6;
	RETURN_CONVEYOR_BUSY	:	UINT  := 7;
END_VAR

(*
	There are two states to the singulation device, releasing and not releasing
	While releasing
		The appropriate grippers are extended:
			- the upsream gripper for all carriers
			- the downstream gripper for racks, totes are detected by the tote sensor at the pin-stop
		When the appropriate grippers are extended (detected using the not-retracted sensor, because the widths of the carriers vary)
			- the pin stop is retracted
			- the downstream photo-eye is monitored for a falling edge to determing if the carrier has exited the singulator
		When the carrier has exited the singulator
			- Releasing is turned off and the state for not releasing is activated
	While not releasing
		The pin stop is extended
		The grippers are retracted when the pin stop is detected in the extended state
		
	The releasing state is enabled when:
		- The distance that the carrier has to travel after exiting the singulator has been traveled by the carrier

	The releasing state is set when:
		- A carrier is detected at the pin stop

	At start-up:
		- the conveyor is not allowed to run
		- all singulation photo-eyes must be clear
			- PE_GrabTrigger, photo-eye at the pin-stop
			- PE_ClearedTrigger, photo-eye downstream of the pin-stop
			- PE_ToteTrigger, photo-eye that detects tote at the pin-stop
		- the device is homed
			- both grippers are retracted to detect home
			- the pin-stop is retracted to detect home
		- after homing, the device is put into a ready state
			- the pin-stop is extended and detected in the extended state
			- the grappers remain retracted are detected in the retracted state
	A release fault is set if it takes too long for a carrier to clear the PE_ClearedTrigger PE (Cfg_TimeOutTime)
	A release can be attempted multiple time (Cfg_RetryLimit). Practically, the release should be attempted once and failed to
		prevent damage to carriers or the specimens they are transporting
	A release fault can only be reset when the device PE's are all clear, to allow a the start-up sequence to be processed
*)

// Process the In_ResetState
rResetState(CLK:=In_ResetState);

// State reset or fault reset clear that current device state and cause the device to start-up again
IF rResetState.Q OR (In_FaultReset AND Out_ReleaseFault) THEN
	// Revert to the StartUp state
	StartUp := TRUE;
	// Revert to the NOT Homed state
	Out_Homed := FALSE;
	tonHomeWait(IN := FALSE);
	// Revert to the NOT Ready state
	Out_Ready := FALSE;
	tonReadyWait(IN := FALSE);
	// Revert to the NOT Running state
	Out_Running := FALSE;
	tonRunningWait(IN := FALSE);

	Out_ReleaseFault := FALSE;
	BadReleaseCount := 0;
	
	Releasing := FALSE;

	// Clear the reset request
	In_ResetState := FALSE;
END_IF

// Use all photo-eyes to determine that the device is clear and can be started up
SingulatorClear := (NOT In_PE_GrabTrigger AND NOT In_PE_ClearedTrigger AND NOT In_PE_ToteTrigger);

// If a start-up is initiated with carriers in the device, set a release fault and cancel the start up
IF StartUp AND NOT SingulatorClear THEN
	Out_ReleaseFault := TRUE;
	StartUp := FALSE;
END_IF

// Home the actuators
IF (StartUp OR NOT Out_Homed OR NOT Out_Ready) AND SingulatorClear THEN
	Status.PAUSED := TRUE;
	
	tonHomeWait.IN := NOT Out_Homed;
	tonHomeWait();

	// Homed is Grabbers retracted and PinStop retracted
	IF NOT Out_Homed THEN
		// Grabber 1
		Grabber_1_Retract := TRUE;
		Grabber_1_Extend := FALSE;
		// Grabber 2
		Grabber_2_Retract := TRUE;
		Grabber_2_Extend := FALSE;
		// PinStop
		PinStop_Retract := TRUE;
		PinStop_Extend := FALSE;
		IF In_Grabber_1_Retracted
		   AND In_Grabber_2_Retracted
		   AND In_PinStop_Retracted
		   THEN
			Out_Homed := tonHomeWait.Q;
		END_IF
	END_IF

	// Ready is Grabbers retracted and PinStop extended
	// All PE's have to be clear for the equipment to be ready
	tonReadyWait.IN := NOT Out_Ready AND Out_Homed AND SingulatorClear;
	tonReadyWait();
	IF NOT Out_Ready AND Out_Homed AND tonReadyWait.IN THEN
		// PinStop
		PinStop_Retract := FALSE;
		PinStop_Extend := TRUE;
		IF In_Grabber_1_Retracted
		   AND In_Grabber_2_Retracted
		   AND In_PinStop_Extended
		   THEN
			Out_Ready := tonReadyWait.Q;
		END_IF
	END_IF

	StartUp := NOT Out_Homed OR NOT Out_Ready;
	Out_Running := FALSE;
	BadReleaseCount := 0;
	Out_ReleaseFault := FALSE;
	Releasing := FALSE;

ELSIF NOT Out_Running THEN

	// Run a timer when the conveyor is running to allow the conveyor to be up-to-speed before actuating any devices
	tonRunningWait.IN := NOT OUT_Running AND Out_Ready AND Out_Homed AND In_ConveyorRunning;
	tonRunningWait();
	Out_Running := tonRunningWait.Q;

	// When Out_Running is turned on, capture the encoder count to allow the release of product when it is detected	
	IF Out_Running THEN
		ClearedPECount := In_EncoderCount;
		Status.PRODUCT_PRESENT := FALSE;
	END_IF
	
ELSIF Out_Running THEN
	Status.PAUSED := FALSE;
	
	// Request to Hold all items
	// Allows external control of the release according to programmed conditions
	IF In_Hold_Request THEN
		// When the pin stop is extended, turn on that the singlulator is holding
		IF In_PinStop_Extended THEN
			Out_Holding := TRUE;
		END_IF
	ELSE
		Out_Holding := FALSE;
	END_IF

	// Singulation Distance Check
	IF In_EncoderCount > ClearedPECount THEN
		ClearedDistance := In_EncoderCount - ClearedPECount;
		RolloverDetect := 0;
	ELSE
		// If the encoder rolls to 0, capture the last distance as an offset
		IF RolloverDetect = 0 THEN
			RolloverDetect := ClearedDistance;
		END_IF
		// The new distance to check is the number of pulses from the Cleared count to the rollover (RolloverDetect)
		// 	plus the current encoder count
		ClearedDistance := RolloverDetect + In_EncoderCount;
	END_IF

	// Release After Distance Requirement is satisfied
	IF ClearedDistance > Cfg_GappingDistance AND NOT Status.PRODUCT_PRESENT THEN
		// Use bit 1 to indicate that the required distance has been cleared to allow the next carrier to be released
		Status.PRODUCT_PRESENT := TRUE;
	END_IF

	// When "PRODUCT_PRESENT" which means that the release distance has been met
	// 	begin to process the RELEASING status
	IF Status.PRODUCT_PRESENT THEN
		// Test for the Holding State
		// Prevent transtion to Releasing while in the holding state
		IF NOT Out_Holding THEN
			// Trigger Releasing when the grab PE is blocked
			IF In_PE_GrabTrigger THEN
				Releasing := TRUE;
			END_IF
		END_IF	
	END_IF

	// Watch release and pin-stop state to make sure product comes through, run timer if not
	ReleaseTimeOut(IN:= Releasing AND In_PinStop_Retracted, PT:= Cfg_TimeOutTime, Q=> , ET=> );

	// Watch for released cleared PE
	// This is a falling-edge trigger that will go true when the cleard photo-eye is blocked
	//	and go false when the cleared photo-eye is cleared
	// Releasing has to remain on while waiting for the cleared trigger photo-eye to transitino
	ClearedTriggerPE(CLK:= (Releasing AND In_PE_ClearedTrigger));

(*	Clearing the photo-eye will:
		- Clear the bad release count
		- Set the In_Encoder count to test for the next release
		- Transition OUT of the releasing state
*)
	IF ClearedTriggerPE.Q THEN
		BadReleaseCount := 0;
		ClearedPECount := In_EncoderCount;
		ClearedDistance := 0;
		Releasing := FALSE;
		Status.PRODUCT_PRESENT := FALSE;
(*
	If the release times out, the BadReleaseCount will be incremented
	In the subsequent code, a non-zero bad release count that exceeds the release attempt limit will set a release fault
	The release fault can only be reset when the device photo-eyes are clear and the reset in issued
	The reset will cause the device to enter its start-up state and home and ready itself
*)
	ELSIF ReleaseTimeOut.Q THEN
		BadReleaseCount := BadReleaseCount + 1;
	END_IF

	// When the Cfg_RetryLimit is exceeded, set the fault
	// This retry limit should always be zero to prevent damage to carriers and specimen because the carrier may be in the path of the 
	// pin-stop
	// Setting the fault does not change the releasing state to prevent carrier/specimen damage and requires the device to be reset
	IF BadReleaseCount >= Cfg_RetryLimit THEN
		Out_ReleaseFault := TRUE;
	END_IF

	// Retry release if Bad release
	// This process originally reset the grippers and pin-stop, along with clearing the releasing state
	// It now only allows an X multiplier of the TimeOutTime for a longer release attempt
	// Actuating the pin-stop could damage carriers/specimen and was disabled
	BadReleaseRetry := (BadReleaseCount > 0) AND (BadReleaseCount <> BadReleaseCount_Old) AND NOT Out_ReleaseFault;
	BadReleaseReTryTimer(IN:= BadReleaseRetry, PT:= T#1S);
	IF BadReleaseReTryTimer.Q THEN
		BadReleaseCount_Old := BadReleaseCount;
	END_IF

ELSE
	// When we aren't detecting any valid state above, turn off Releasing to extend the grippers until the pin-stop is extended
	// This should never be executed but is here just-in-case
	// NOT Out_Running should catch all unknown states and prevent the transition to Out_Running based on the homed and ready states
	Releasing := FALSE;
END_IF

// Only process if we are Ready
// Actuation is controlled for all other states during start-up
IF Out_Ready THEN
	// Test for Releasing and actuate accordingly and pause request
	// In_Pause and In_Hold_Request perform the samd function, but at different stages of the process
	// In_Pause affect the system when it is releasing
	// In_Hold prevent the system from transitioning into the Releasing state
	IF Releasing AND NOT In_Pause THEN
		// Grabber 1 - Always Extend
		Grabber_1_Retract := FALSE;
		Grabber_1_Extend := TRUE;
		// Grabber 2 - Extend only when a tote is not detected
		IF In_PE_ToteTrigger THEN
			Grabber_2_Retract := TRUE;
			Grabber_2_Extend := FALSE;
		ELSE
			Grabber_2_Retract := FALSE;
			Grabber_2_Extend := TRUE;
		END_IF
		// Only process the pin-stop when the gripper(s) are not in the retracted state
		// Only check grabber 1 because grabber 2 could remain retracted for a tote
		IF NOT In_Grabber_1_Retracted THEN
			// PinStop retract when the grippers are holding
			PinStop_Retract := TRUE;
			PinStop_Extend := FALSE;
		END_IF
	// When not releasing, only actuate the pin-stop when the device is clear to prevent damage to carriers and/or specimen
	ELSE
		IF SingulatorClear THEN
			// PinStop extend when the device is clear
			PinStop_Retract := FALSE;
			PinStop_Extend := TRUE;
			// Only process the grabbers when the pin-stop is in the extended state
			IF In_PinStop_Extended THEN
				// Grabber 1 - Always Retract
				Grabber_1_Retract := TRUE;
				Grabber_1_Extend := FALSE;
				// Grabber 2 - Always Retract
				Grabber_2_Retract := TRUE;
				Grabber_2_Extend := FALSE;
			END_IF
		// When the device is not clear and we are not releasing, extend both grabbers when the pin-stop is not extended
		ELSE
			IF In_PinStop_Retracted THEN
				// Grabber 1 - Always Extend when the singulator is not clear
				Grabber_1_Retract := FALSE;
				Grabber_1_Extend := TRUE;
				// Grabber 2 - Always Extend when the singulator is not clear
				Grabber_2_Retract := FALSE;
				Grabber_2_Extend := TRUE;
			ELSE
				Grabber_1_Retract := TRUE;
				Grabber_1_Extend := FALSE;
				Grabber_2_Retract := TRUE;
				Grabber_2_Extend := FALSE;
			END_IF
		END_IF
	END_IF
END_IF

// Activate all the outputs in one place
Status_Output.GRABBER_1_OCCUPIED := Grabber1(Active := In_Grabber_1_Auto, Extend:= Grabber_1_Extend, Retract := Grabber_1_Retract);
Status_Output.GRABBER_2_OCCUPIED := Grabber2(Active := In_Grabber_2_Auto, Extend:= Grabber_2_Extend, Retract := Grabber_2_Retract);
Status_Output.PINSTOP_OUT := PinStop(Active:= In_PinStop_Auto, Extend := PinStop_Extend, Retract:= PinStop_Retract);

ACTION a_HoldProduct:
	// Grabber 1
	Grabber_1_Retract := FALSE;
	Grabber_1_Extend := TRUE;
	
	// Grabber 2
	Grabber_2_Retract := FALSE;
	Grabber_2_Extend := TRUE;
END_ACTION

ACTION a_ResetGrabbers:
// Grabber 1 Retract
Grabber_1_Retract := TRUE;
Grabber_1_Extend := FALSE;
// Grabber 2 Retract
Grabber_2_Retract := TRUE;
Grabber_2_Extend := FALSE;
// PinStop Extend
PinStop_Retract := FALSE;
PinStop_Extend := TRUE;
// Reset Releasing
Releasing := FALSE;
END_ACTION

METHOD Grabber1 : BOOL
VAR_INPUT
	Active	: BOOL;	
	Extend	: BOOL;
	Retract	: BOOL;
END_VAR
IF Active THEN
	IF Extend THEN
		Out_Grabber_1_Ext := TRUE;
		Out_Grabber_1_Ret := FALSE;
	ELSIF Retract THEN
		Out_Grabber_1_Ext := FALSE;
		Out_Grabber_1_Ret := TRUE;
	ELSE
		Out_Grabber_1_Ext := FALSE;
		Out_Grabber_1_Ret := FALSE;
	END_IF
ELSE
	Out_Grabber_1_Ext := FALSE;
	Out_Grabber_1_Ret := FALSE;
END_IF

Grabber1 := Out_Grabber_1_Ext OR In_Grabber_1_Extended;
END_METHOD

METHOD Grabber2 : BOOL
VAR_INPUT
	Active	: BOOL;	
	Extend	: BOOL;
	Retract	: BOOL;
END_VAR
IF Active THEN
	IF Extend THEN
		Out_Grabber_2_Ext := TRUE;
		Out_Grabber_2_Ret := FALSE;
	ELSIF Retract THEN
		Out_Grabber_2_Ext := FALSE;
		Out_Grabber_2_Ret := TRUE;
	ELSE
		Out_Grabber_2_Ext := FALSE;
		Out_Grabber_2_Ret := FALSE;
	END_IF
ELSE
	Out_Grabber_2_Ext := FALSE;
	Out_Grabber_2_Ret := FALSE;
END_IF

Grabber2 := Out_Grabber_2_Ext OR In_Grabber_2_Extended;
END_METHOD

METHOD PinStop : BOOL
VAR_INPUT
	Active	: BOOL;	
	Extend	: BOOL;
	Retract	: BOOL;
END_VAR
IF Active THEN
	IF Extend THEN
		Out_PinStop_Ext := TRUE;
		Out_PinStop_Ret := FALSE;
	ELSIF Retract THEN
		Out_PinStop_Ext := FALSE;
		Out_PinStop_Ret := TRUE;
	ELSE
		Out_PinStop_Ext := FALSE;
		Out_PinStop_Ret := FALSE;
	END_IF
ELSE
	Out_PinStop_Ext := FALSE;
	Out_PinStop_Ret := FALSE;
END_IF

PinStop := Out_PinStop_Ext OR In_PinStop_Extended;
END_METHOD

END_FUNCTION_BLOCK

// ---- POUs/Sorter.TcPOU
PROGRAM Sorter
VAR
	nSorterClearIdx				: DINT;
	bSimulate					: BOOL := FALSE;	// Indicates when runing a simulation
//----------------------------------------P2140--------------------------------------------------------------	
	st_ToInduct_P2140					: ST_ItemTemporary;	// This is the next item to be inducted onto the sorter
	st_Inducting_P2140				: ST_ItemTemporary;	// This is the next item to be inducted onto the sorter
	st_InductUpdate_P2140				: ST_ItemTemporary;	// This is to update an item already being inducted
	st_Sorter_P2140					: ST_Sorter;
	aSorterDiverts_P2140 				: ARRAY[DIVERTMIN_P2140..NUMBEROFDIVERTS_P2140] OF ST_Divert;

	st_SorterEncoder_P2140 			: ST_Encoder;
	fb_SorterEncoder_P2140 			: FB_ProcessEncoder;

	tEncoderOK_P2140			: TON;
	nLastEncoderCount_P2140	: UDINT;

	fb_CommissionSorterDiverts_P2140	: FB_DivertCommission;
	st_TempItem_P2140					: ST_ItemTemporary;	// Store temporary Item info until BCR data is received
	SorterDischargeItem_P2140			: ST_Item;	// Last Item discharged from the end of the sorter

	DivertToCommission_P2140			: UINT := 0;	// Non-zero value will send all items to this divert

	{attribute 'OPC.UA.DA' := '0'}
	P2140_SorterLog				:	FB_SorterLog;
	P2140_DivertLog				:	FB_DivertLog;	

	sMessage			: STRING;

	ClearSorterArray	: BOOL;
//----------------------------------------P2150--------------------------------------------------------------	
	st_ToInduct_P2150					: ST_ItemTemporary;	// This is the next item to be inducted onto the sorter
	st_Inducting_P2150				: ST_ItemTemporary;	// This is the next item to be inducted onto the sorter
	st_InductUpdate_P2150				: ST_ItemTemporary;	// This is to update an item already being inducted
	st_Sorter_P2150					: ST_Sorter;
	aSorterDiverts_P2150 				: ARRAY[DIVERTMIN_P2150..NUMBEROFDIVERTS_P2150] OF ST_Divert;

	st_SorterEncoder_P2150 			: ST_Encoder;
	fb_SorterEncoder_P2150 			: FB_ProcessEncoder;

	tEncoderOK_P2150			: TON;
	nLastEncoderCount_P2150	: UDINT;

	fb_CommissionSorterDiverts_P2150	: FB_DivertCommission;

	st_TempItem_P2150					: ST_ItemTemporary;	// Store temporary Item info until BCR data is received
	SorterDischargeItem_P2150			: ST_Item;	// Last Item discharged from the end of the sorter

	DivertToCommission_P2150			: UINT := 0;	// Non-zero value will send all items to this divert

	{attribute 'OPC.UA.DA' := '0'}
	P2150_SorterLog				:	FB_SorterLog;
	P2150_DivertLog				:	FB_DivertLog;	
END_VAR

VAR PERSISTENT
//----------------------------------------P2140--------------------------------------------------------------		
	aSorterItems_P2140 				: ARRAY[SORTERENCODERMIN_P2140..SORTERENCODERMAX_P2140] OF ST_Item;	// Persist the Items to Sort array
	st_Sorter_P2140Cfg				: ST_SorterConfig; 	// Persist Sorter configuration
	aSorterDiverts_P2140Cfgs 		: ARRAY[DIVERTMIN_P2140..NUMBEROFDIVERTS_P2140] OF ST_DivertCfg; 	// Persist Sorter Configuration
//----------------------------------------P2150--------------------------------------------------------------		
	aSorterItems_P2150 				: ARRAY[SORTERENCODERMIN_P2150..SORTERENCODERMAX_P2150] OF ST_Item;	// Persist the Items to Sort array
	st_Sorter_P2150Cfg				: ST_SorterConfig; 	// Persist Sorter configuration
	aSorterDiverts_P2150Cfgs 		: ARRAY[DIVERTMIN_P2150..NUMBEROFDIVERTS_P2150] OF ST_DivertCfg; 	// Persist Sorter Configuration
END_VAR

VAR CONSTANT
//----------------------------------------P2140--------------------------------------------------------------	
	SORTERMASKSIZE_P2140				: UINT := 12;		// Number of bits to mask into the Encoder Count, will define the size of the SORTERENCODERMAX value
	{attribute 'OPC.UA.DA' := '1'}
	NUMBEROFDIVERTS_P2140				: DINT := 2;
	DIVERTMIN_P2140					: DINT := 1;
	{attribute 'OPC.UA.DA' := '1'}
	SORTERENCODERMAX_P2140			: UDINT := ((LREAL_TO_UDINT(EXPT(2,SORTERMASKSIZE_P2140)))-1); // Calculated size based on the bitmask 
	{attribute 'OPC.UA.DA' := '1'}
	SORTERENCODERMIN_P2140			: UDINT := 0;
//----------------------------------------P2150--------------------------------------------------------------	
	SORTERMASKSIZE_P2150				: UINT := 11;		// Number of bits to mask into the Encoder Count, will define the size of the SORTERENCODERMAX value
	{attribute 'OPC.UA.DA' := '1'}
	NUMBEROFDIVERTS_P2150				: DINT := 5;
	DIVERTMIN_P2150					: DINT := 1;
	{attribute 'OPC.UA.DA' := '1'}
	SORTERENCODERMAX_P2150			: UDINT := ((LREAL_TO_UDINT(EXPT(2,SORTERMASKSIZE_P2150)))-1); // Calculated size based on the bitmask 
	{attribute 'OPC.UA.DA' := '1'}
	SORTERENCODERMIN_P2150			: UDINT := 0;
	
END_VAR

// Sorter clear when the system is restarted or downloaded (INIT=TRUE for first scan)
IF (GVL_IO.INIT AND NOT st_Sorter_P2140Cfg.RetainOnRestart) OR ClearSorterArray THEN
	FOR nSorterClearIdx := UDINT_TO_DINT(SORTERENCODERMIN_P2140) TO UDINT_TO_DINT(SORTERENCODERMAX_P2140) BY 1 DO
		IF nSorterLogEnable.SORTER_DUMP THEN
			IF aSorterItems_P2140[nSorterClearIdx].ID <> '' THEN
				IF .nSorterLogEnable.SORTER_DUMP THEN
					sMessage := CONCAT(' Item: ', aSorterItems_P2140[nSorterClearIdx].ID);
					sMessage := CONCAT(sMessage,' Index: ');
					sMessage := CONCAT(sMessage, DINT_TO_STRING(nSorterClearIdx));
					// Write to the Error List
					ADSLOGSTR( msgCtrlMask := ADSLOG_MSGTYPE_HINT OR ADSLOG_MSGTYPE_LOG
						, msgFmtStr := 'P2140 Array Dump Info: %s'
						, strArg := sMessage);
				END_IF
			END_IF
		END_IF
		aSorterItems_P2140[nSorterClearIdx] := BlankItem;
	END_FOR
	ClearSorterArray := FALSE;
END_IF

// Setup and process the Sorter Encoder
st_SorterEncoder_P2140.EncoderRawCount := GVL_IO.ENC_9031_Raw;
st_SorterEncoder_P2140.BitMaskSize := SORTERMASKSIZE_P2140;
fb_SorterEncoder_P2140(Encoder := st_SorterEncoder_P2140, Simulate := bSimulate);
(*
	Initialize Diverts here. 
	Tie variables commented IO to physical IO address
*)
//Divert #1
aSorterDiverts_P2140[1].Config := aSorterDiverts_P2140Cfgs[1];
aSorterDiverts_P2140[1].ConfirmPE := Photoeyes.PE_10302.Out; 			
aSorterDiverts_P2140[1].FullPE := Photoeyes.PE_10302.Out_OnFltrd;   			

//Divert #2
aSorterDiverts_P2140[2].Config := aSorterDiverts_P2140Cfgs[2];
aSorterDiverts_P2140[2].ConfirmPE := Photoeyes.PE_10151.Out AND NOT Solenoids.PL2140_01.In_EquipRtrcdFdbck;	
aSorterDiverts_P2140[2].FullPE := Photoeyes.PE_10091.Out_OnFltrd;

fb_CommissionSorterDiverts_P2140(
			InductTrigger := Photoeyes.PE_10081.Out,
			ReferenceValue := st_SorterEncoder_P2140.CurrentCount, 
			DischargeTrigger := Photoeyes.PE_10091.Out_OffFltrd,
			TestTime := T#10S, Diverts := aSorterDiverts_P2140);

// Provide a "hard-coded" default destination.
IF st_Sorter_P2140Cfg.DefaultDestination <= 0 THEN
	st_Sorter_P2140Cfg.DefaultDestination := 1;
END_IF						

// Check for a changed Default Destination from the messaging
IF P2140_DefaultDestination <> 0
   AND P2140_DefaultDestination <> st_Sorter_P2140Cfg.DefaultDestination
   THEN
   	st_Sorter_P2140Cfg.DefaultDestination := DINT_TO_UINT(P2140_DefaultDestination);
END_IF

// Name of the sorter equipment
st_Sorter_P2140Cfg.Name := Conveyors.cfgP2140Label;
st_Sorter_P2140Cfg.DivertCount := NUMBEROFDIVERTS_P2140;
IF DivertToCommission_P2140 > 0 THEN
	st_Sorter_P2140Cfg.DefaultDestination := DivertToCommission_P2140;
END_IF
st_Sorter_P2140.EncoderCounts := st_SorterEncoder_P2140.CurrentCount;
st_Sorter_P2140.InductPE := PhotoEyes.PE_10081.Out_OnOffFltrd;
st_Sorter_P2140.DischargePE := Photoeyes.PE_10091.Out;

// Test the Encoder
tEncoderOK_P2140.IN := (Conveyors.P2140_Status.Sts_IsRunning AND (st_Sorter_P2140.EncoderCounts = nLastEncoderCount_P2140));
nLastEncoderCount_P2140 := st_Sorter_P2140.EncoderCounts;
tEncoderOK_P2140(PT:=T#1S);

// OK when Q is not on, but the alarm is reversed
  GVL_IO.ENC_9031_OK := tEncoderOK_P2140.Q;
  
// Publish the sorter name
  GVL_IO.Sorter_P2140Name := st_Sorter_P2140Cfg.Name;

// Sorter
(*
	ProcessBuffers processes all associated buffers (Sorter/Divert/Arrival/Transport/Update)
	Items arriving at the sorter are detected and processed in this function block then deliverd to the SorterProgram
	Items inducted into sorter produce TransportResponse messages in this function block
	Items diverted off the sorter produce TransportComplete messages in this function block
*)
ProcessBuffers_P2140(st_NextToInduct := st_ToInduct_P2140
				, st_TempInductItem := st_TempItem_P2140
				, st_UpdateItem := st_Inducting_P2140
				, st_Sorter := st_Sorter_P2140
				, aDiverts := aSorterDiverts_P2140
				, aItems := aSorterItems_P2140
				, DivertToCommission := DivertToCommission_P2140
				,ItemsArrayMin := SORTERENCODERMIN_P2140
				,ItemsArrayMax := SORTERENCODERMAX_P2140
				,DefaultDestIdx => st_Sorter_P2140Cfg.DefaultDestIdx
				,RecircDestIdx => st_Sorter_P2140Cfg.RecircDestIdx);

// Sorter LOG logs induct/discharge PE's and prepares the Temporory Record for unidentified items
P2140_SorterLog(
				SorterToLog := st_Sorter_P2140,
				SorterLogEnable := .nSorterLogEnableP2140,
				ToInduct := st_ToInduct_P2140,
				TempItem => );

IF P2140_SorterLog.TempItem.Item.ID <> '' THEN
	IF P2140_SorterLog.TempItem.Item.ID <> st_TempItem_P2140.Item.ID THEN
		st_TempItem_P2140 := P2140_SorterLog.TempItem;
	END_IF
END_IF

(*
	SorterProgram is a separate Program
	Config portion of the st_sorter is separate to allow it be be persistent.
*)
st_sorter_P2140.Config := st_sorter_P2140Cfg;
Sorter_P2140(st_Sorter := st_Sorter_P2140
		, In_ItemToInduct := st_ToInduct_P2140.Item
		, In_InductingItem := st_Inducting_P2140.Item
		, aItems := aSorterItems_P2140
		, aDiverts := aSorterDiverts_P2140
		, st_tempItem := st_TempItem_P2140
		, ItemsArrayMax := SORTERENCODERMAX_P2140
		, ItemsArrayMin := SORTERENCODERMIN_P2140
		, DivertArrayMax := NUMBEROFDIVERTS_P2140
		, DivertArrayMin := DIVERTMIN_P2140
		, st_DischargeItem => SorterDischargeItem_P2140);

// Log the diverts
P2140_DivertLog(DivertArray := aSorterDiverts_P2140,
				DivertLogEnable := .nDivertLogEnableP2140,
				EncoderCounts := st_SorterEncoder_P2140.CurrentCount);

//--------------------------------------Sorter P2150------------------------------------------	

// Sorter clear when the system is restarted or downloaded (INIT=TRUE for first scan)
IF (GVL_IO.INIT AND NOT st_Sorter_P2150Cfg.RetainOnRestart) OR ClearSorterArray THEN
	FOR nSorterClearIdx := UDINT_TO_DINT(SORTERENCODERMIN_P2150) TO UDINT_TO_DINT(SORTERENCODERMAX_P2150) BY 1 DO
		IF nSorterLogEnable.SORTER_DUMP THEN
			IF aSorterItems_P2150[nSorterClearIdx].ID <> '' THEN
				IF .nSorterLogEnable.SORTER_DUMP THEN
					sMessage := CONCAT(' Item: ', aSorterItems_P2150[nSorterClearIdx].ID);
					sMessage := CONCAT(sMessage,' Index: ');
					sMessage := CONCAT(sMessage, DINT_TO_STRING(nSorterClearIdx));
					// Write to the Error List
					ADSLOGSTR( msgCtrlMask := ADSLOG_MSGTYPE_HINT OR ADSLOG_MSGTYPE_LOG
						, msgFmtStr := 'P2150 Array Dump Info: %s'
						, strArg := sMessage);
				END_IF
			END_IF
		END_IF
		aSorterItems_P2150[nSorterClearIdx] := BlankItem;
	END_FOR
	ClearSorterArray := FALSE;
END_IF

// Setup and process the Sorter Encoder
st_SorterEncoder_P2150.EncoderRawCount := GVL_IO.ENC_9091_Raw;
st_SorterEncoder_P2150.BitMaskSize := SORTERMASKSIZE_P2150;
fb_SorterEncoder_P2150(Encoder := st_SorterEncoder_P2150, Simulate := bSimulate);

(*
	Initialize Diverts here. 
	Tie variables commented IO to physical IO address
*)

//Divert #1
aSorterDiverts_P2150[1].Config := aSorterDiverts_P2150Cfgs[1];
aSorterDiverts_P2150[1].ConfirmPE := Photoeyes.PE_3231.Out; 			
aSorterDiverts_P2150[1].FullPE := Photoeyes.PE_3231.Out;   			

//Divert #2
aSorterDiverts_P2150[2].Config := aSorterDiverts_P2150Cfgs[2];
aSorterDiverts_P2150[2].ConfirmPE := Photoeyes.PE_3111.Out; 		
aSorterDiverts_P2150[2].FullPE := Photoeyes.PE_3111.Out;   		

//Divert #3 
aSorterDiverts_P2150[3].Config := aSorterDiverts_P2150Cfgs[3];
aSorterDiverts_P2150[3].ConfirmPE := Photoeyes.PE_4201.Out; 		
aSorterDiverts_P2150[3].FullPE := Photoeyes.PE_4201.Out;   	

//Divert #4 
aSorterDiverts_P2150[4].Config := aSorterDiverts_P2150Cfgs[4];
aSorterDiverts_P2150[4].ConfirmPE := Photoeyes.PE_4091.Out; 		
aSorterDiverts_P2150[4].FullPE := Photoeyes.PE_4091.Out; 

//Divert #5
aSorterDiverts_P2150[5].Config := aSorterDiverts_P2150Cfgs[5];
aSorterDiverts_P2150[5].ConfirmPE := Photoeyes.PE_4161.Out; 		
aSorterDiverts_P2150[5].FullPE := Photoeyes.PE_4161.Out; 	

fb_CommissionSorterDiverts_P2150(
			InductTrigger := Photoeyes.PE_2131.Out,
			ReferenceValue := st_SorterEncoder_P2150.CurrentCount, 
			DischargeTrigger := Photoeyes.PE_4161.Out_OffFltrd,
			TestTime := T#10S, Diverts := aSorterDiverts_P2150);

// Provide a "hard-coded" default destination.
IF st_Sorter_P2150Cfg.DefaultDestination <= 0 THEN
	st_Sorter_P2150Cfg.DefaultDestination := 30;
END_IF						

// Check for a changed Default Destination from the messaging
IF P2150_DefaultDestination <> 0
   AND P2150_DefaultDestination <> st_Sorter_P2150Cfg.DefaultDestination
   THEN
   	st_Sorter_P2150Cfg.DefaultDestination := DINT_TO_UINT(P2150_DefaultDestination);
END_IF

// Name of the sorter equipment
st_Sorter_P2150Cfg.Name := Conveyors.cfgP2150Label;
st_Sorter_P2150Cfg.DivertCount := NUMBEROFDIVERTS_P2150;
IF DivertToCommission_P2150 > 0 THEN
	st_Sorter_P2150Cfg.DefaultDestination := DivertToCommission_P2150;
END_IF
st_Sorter_P2150.EncoderCounts := st_SorterEncoder_P2150.CurrentCount;
st_Sorter_P2150.InductPE := PhotoEyes.PE_2131.Out_OffFltrd;
st_Sorter_P2150.DischargePE := Photoeyes.PE_4161.Out;

// Test the Encoder
tEncoderOK_P2150.IN := (Conveyors.P2150_Status.Sts_IsRunning AND (st_Sorter_P2150.EncoderCounts = nLastEncoderCount_P2150));
nLastEncoderCount_P2150 := st_Sorter_P2150.EncoderCounts;
tEncoderOK_P2150(PT:=T#1S);

// OK when Q is not on, but the alarm is reversed
  GVL_IO.ENC_9091_OK := tEncoderOK_P2150.Q;
  
// Publish the sorter name
  GVL_IO.Sorter_P2150Name := st_Sorter_P2150Cfg.Name;

// Sorter
(*
	ProcessBuffers processes all associated buffers (Sorter/Divert/Arrival/Transport/Update)
	Items arriving at the sorter are detected and processed in this function block then deliverd to the SorterProgram
	Items inducted into sorter produce TransportResponse messages in this function block
	Items diverted off the sorter produce TransportComplete messages in this function block
*)
ProcessBuffers_P2150(st_NextToInduct := st_ToInduct_P2150
				, st_TempInductItem := st_TempItem_P2150
				, st_UpdateItem := st_Inducting_P2150
				, st_Sorter := st_Sorter_P2150
				, aDiverts := aSorterDiverts_P2150
				, aItems := aSorterItems_P2150
				, DivertToCommission := DivertToCommission_P2150
				,ItemsArrayMin := SORTERENCODERMIN_P2150
				,ItemsArrayMax := SORTERENCODERMAX_P2150
				,DefaultDestIdx => st_Sorter_P2150Cfg.DefaultDestIdx
				,RecircDestIdx => st_Sorter_P2150Cfg.RecircDestIdx);

// Sorter log logs induct/discharge PE's and prepares the Temporory Record for unidentified items
P2150_SorterLog(
				SorterToLog := st_Sorter_P2150,
				SorterLogEnable := .nSorterLogEnableP2150,
				ToInduct := st_ToInduct_P2150,
				TempItem => );

IF P2150_SorterLog.TempItem.Item.ID <> '' THEN
	IF P2150_SorterLog.TempItem.Item.ID <> st_TempItem_P2150.Item.ID THEN
		st_TempItem_P2150 := P2150_SorterLog.TempItem;
	END_IF
END_IF

(*
	SorterProgram is a separate Program
	Config portion of the st_sorter is separate to allow it be be persistent.
*)
st_sorter_P2150.Config := st_sorter_P2150Cfg;
Sorter_P2150(st_Sorter := st_Sorter_P2150
		, In_ItemToInduct := st_ToInduct_P2150.Item
		, In_InductingItem := st_Inducting_P2150.Item
		, aItems := aSorterItems_P2150
		, aDiverts := aSorterDiverts_P2150
		, st_tempItem := st_TempItem_P2150
		, ItemsArrayMax := SORTERENCODERMAX_P2150
		, ItemsArrayMin := SORTERENCODERMIN_P2150
		, DivertArrayMax := NUMBEROFDIVERTS_P2150
		, DivertArrayMin := DIVERTMIN_P2150
		, st_DischargeItem => SorterDischargeItem_P2150);

// Log the diverts
P2150_DivertLog(DivertArray := aSorterDiverts_P2150,
				DivertLogEnable := .nDivertLogEnableP2150,
				EncoderCounts := st_SorterEncoder_P2150.CurrentCount);

END_PROGRAM

// ---- FunctionBlocks/Encoder/FB_ProcessEncoder.TcPOU
FUNCTION_BLOCK FB_ProcessEncoder
VAR_IN_OUT
	Encoder:	ST_Encoder;
END_VAR
VAR_INPUT
	Simulate:	BOOL;	// Return a Simulate count
	SimPulseInterval: TIME := T#1S; // Time between simulated encoder pulses
END_VAR
VAR
	//Simulation Variables
	SimEncoderTimer		: TON;	// Timer used to simulate encoder movement
	sEncoderString		: STRING;	// Current Encoder Count formatted as a string
END_VAR

(*
	The Beckhoff encoder card cannot be configured to roll-over at a specfic interval, therefore it must be
	bitWise AND masked to approximate the size of the sorter array to maintain a 1-1 encoder pulse to sorter array index relationship.
	The masking is accomplished by calculating (2^n - 1) where (2^n - 1) is greater than the length of the sorter in pulses.
	The "- 1" flips all the bits to the right of the 2^n value. When this is ANDED with the encoder count, the count effectively
	"rolls over" when the 2^n value is reached. The encoder count will continue to increase to the maximum value (UINT[65535] UDINT[4294967295],
	but 0 to (2^n - 1) will be the effective range of the encoder.

	65535 AND 0 [(2^0) - 1] = 0			65535 / 255 [(2^8) - 1] = 255
	65535 AND 1 [(2^1) - 1] = 1			65535 / 511 [(2^9) - 1] = 511
	65535 AND 3 [(2^2) - 1] = 3			65535 / 1023 [(2^10) - 1] = 1023
	65535 AND 7 [(2^3) - 1] = 7			65535 / 2047 [(2^11) - 1] = 2047
	65535 AND 15 [(2^4) - 1] = 15		65535 / 4095 [(2^12) - 1] = 4095
	65535 AND 31 [(2^5) - 1] = 31		65535 / 8191 [(2^13) - 1] = 8191
	65535 AND 63 [(2^6) - 1] = 63		65535 / 16383 [(2^14) - 1] = 16383
	65535 AND 127 [(2^7) -1] = 127		65535 / 32767 [(2^15) - 1] = 32767
	                       				65535 / 65535 [(2^16) - 1] = 65535

*)

SimEncoderTimer(IN := Simulate, PT := SimPulseInterval);
IF Simulate THEN
	IF SimEncoderTimer.Q THEN
		Encoder.CurrentCount := Encoder.CurrentCount + 1;
		IF Encoder.CurrentCount >= LREAL_TO_UDINT(EXPT(2,Encoder.BitMaskSize)) THEN
			Encoder.CurrentCount := 0;
		END_IF
		// Reset the Timer
		SimEncoderTimer(IN := FALSE, PT := SimPulseInterval);
	END_IF
ELSE
	Encoder.CurrentCount := Encoder.EncoderRawCount AND (LREAL_TO_UDINT(EXPT(2,Encoder.BitMaskSize)) - 1);
END_IF

// Front and Rear space padding on the current encoder count
Encoder.EncoderString := CONCAT(' ',UDINT_TO_STRING(Encoder.CurrentCount));
Encoder.EncoderString := CONCAT(Encoder.EncoderString, ' ');

END_FUNCTION_BLOCK

// ---- FunctionBlocks/Divert/Functions/FB_DivertCommission.TcPOU
FUNCTION_BLOCK FB_DivertCommission
VAR_INPUT
	InductTrigger	: BOOL; //This is the starting point you want to measure from
	ReferenceValue 	: UDINT; //This is the measurement reference you want to use (most typically will be an encoder value)
	DischargeTrigger: BOOL; //This is the end point that you want to stop measuring
	Reset			: BOOL; //1 - reset all values 0 - keep existing values
	TestTime 		: TIME; //Maximum amount of time it could possibly take to get measurement. If you're not getting a measurement, increase this time
END_VAR

VAR_IN_OUT
	Diverts			: ARRAY[*] OF ST_Divert; //Diverts that you want to measure
END_VAR

VAR
	DivertIndex		: DINT;
	StartCount 		: UDINT;
	EndCount 		: UDINT;
	InductFlag		: BOOL;
	NumberofDiverts	: DINT; 
	DivertLength 	: ARRAY[0..16] OF UDINT;
	DivertTime 		: ARRAY[0..16] OF TIME;
	DischargeFlag	: ARRAY[0..16] OF BOOL;
	
	DivertTimer 	: TON := (PT := TestTime);	
END_VAR

DivertTimer();

NumberofDiverts	:= UPPER_BOUND(Diverts,1);

IF NumberofDiverts < 17 THEN
	IF InductTrigger AND NOT InductFlag THEN
		StartCount := ReferenceValue;
		DivertTimer(IN := TRUE);
		InductFlag := TRUE;
	END_IF
	
	IF DischargeTrigger AND NOT DischargeFlag[0] THEN
		DivertLength[0] := ReferenceValue;
		DivertTime[0]   := DivertTimer.ET;
		DivertTimer(IN := FALSE);
		DischargeFlag[0] := TRUE;
	END_IF
	
	FOR DivertIndex := 1 TO NumberOfDiverts DO
		IF Diverts[DivertIndex].ConfirmPE AND NOT DischargeFlag[DivertIndex] THEN
			DivertLength[DivertIndex]  := ReferenceValue;
			DivertTime[DivertIndex]    := DivertTimer.ET;
			DischargeFlag[DivertIndex] := TRUE;	
		END_IF
	END_FOR
	
	IF Reset THEN
		InductFlag := FALSE;
		DivertTimer(IN := FALSE);
		FOR DivertIndex := 0 TO NumberOfDiverts DO
			DischargeFlag[DivertIndex] := FALSE;
			DivertLength[DivertIndex] := 0;
		END_FOR
	END_IF
END_IF

END_FUNCTION_BLOCK

